FUNCTION_BLOCK SM_DoorDasher EXTENDS KvalStateMachineBaseExt
VAR_INPUT
	cmd_bReset						: BOOL; // reset from error.
	cmd_bCrossTransfer				: BOOL; // true to start cross transfering between 2 adjacent tables.
	cmd_bInlineTransfer				: BOOL; // true to start inline transfering between 2 adjacent tables.
	cmd_bRotateDoor					: BOOL; // true to rotate the door.
	cmd_bCenterDoor					: BOOL; // true to center the door before rotation.
	cmd_bDoorDash					: BOOL; // true to start transport door between adjacent tables.
	cmd_iSource						: INT; // starting table to cross from.
	cmd_iTarget						: INT; // ending table to cross to.
	pstTable						: POINTER TO SM_TableManager;
	pstDoorTrack					: POINTER TO ST_DoorTrack; // pointer to the TableManager's DoorTrack object.
	itfDoorTracker					: I_DoorTracker;
	
	config_tCrossFeedTargetFenceStopEyeValidTime	: TIME := T#20MS;	// time for a valid target fence table's eye.
	
	config_tCrossFeedTargetEyeValidTime	: TIME := T#20MS;	// debouncing time for a valid target table's eye.
	config_tCrossFeedSourceEyeValidTime	: TIME := T#20MS;
	config_tInlineFeedSourceEyeValidTime	: TIME := T#20MS;
	config_tStopMotorValidTime	: TIME := T#30MS;
	
	config_tCrossFeedTargetEyeRisingPreSearchTime	: TIME := T#0.25S;
	config_tInlineFeedTargetEyeRisingPreSearchTime	: TIME := T#0.25S;
	
	config_tCrossFeedTargetEyeRisingPreValidTime	: TIME := T#20MS;
	config_tInlineFeedTargetEyeRisingValidTime	: TIME := T#2.0S;
	
	config_tCrossFeedTargetEyeRisingPostSearchTime	: TIME := T#2.0S;
	config_tInlineFeedTargetEyeRisingPostSearchTime	: TIME := T#2.0S;
	
	config_tCrossFeedTargetEyeRisingPostValidTime	: TIME := T#20MS;
	config_tInlineFeedTargetEyeRisingPostValidTime	: TIME := T#20MS;
	
	config_tCrossFeedTargetEyeRisingPreMaxTime	: TIME := T#3.0S;
	config_tInlineFeedTargetEyeRisingMaxTime	: TIME := T#3.0S;
	
	config_tCrossFeedTargetEyeRisingPostMaxTime	: TIME := T#5.0S;
	config_tInlineFeedTargetEyeFallingMaxTime	: TIME := T#10.0S;
	config_tCrossFeedWaitForAllDoorDashersReady	: TIME := T#0.25S;
	config_tInlineFeedWaitForAllDoorDashersReady	: TIME := T#0.25S;
	config_tCrossFeedSourceEyeRisingSearchTime	: TIME := T#20MS;
	config_tInlineFeedSourceEyeRisingSearchTime	: TIME := T#20MS;
	config_tFindSourceCrossEyeMaxTimeSec		: TIME := T#2.75S; // timeout for finding source's rising edge of feed eye.
	config_tFindSourceInlineEyeMaxTimeSec		: TIME := T#3.5S; // timeout for finding source's rising edge of feed eye.
	config_fFindTargetEyeTimeSec		: LREAL := 12;	// timeout for finding rising or falling edge of the target table's eye. Assumes source and target tables are adjacent neighbors.
	config_fFindRisingEdgeOfTargetFenceEyeTime		: TIME := T#0.25S;
	config_tInlineTargetFeedEyeFallingEdgeTime	: TIME := T#50MS;

	config_iTableArrayIndex			: INT;		// The array table index.
END_VAR
VAR_OUTPUT		
	bMovingFwd					: BOOL; // true if eSource > eTarget
	bIsTargetBufferTable				: BOOL; // used by inline-transfer seq. True to skip the re-feedin seq to center the door on table if the target table is a buffer table with T1 option, which can only inline-transfer and not (cross-transfer or self-center).  
	bIsConveyorAtTarget			: BOOL; // true if the target table is the conveyor type (C235)	
	bIsConveyorAtSource			: BOOL; // true if the source table is the conveyor type (C235)	
	
	bDoorInMachineAtSource		: BOOL;
	bDoorInMachineAtTarget		: BOOL;
	iStopTableIndex : INT;
	bSourceTrailingNeighborDoorDasherBusy : BOOL;
	bSourceLeadingNeighborDoorDasherBusy : BOOL;
	bAllCrossCylsExtended		: BOOL;
	bAllCrossCylsRetracted		: BOOL;
	bOkToTransferOutDoor 		: BOOL;
	bTransferring				: BOOL;
	bCrossTransferSeqRunning	: BOOL;
	bInlineTransferSeqRunning	: BOOL;
	bFoundTarget				: BOOL;
	bAllSourceAndTargetExternal : BOOL;
	bCenteringDoorStarted		: BOOL;
	bCenteringDoorComplete		: BOOL;
	bAnyTableExternal 			: BOOL;
	bSourceTableReady			: BOOL;
	bAllTablesReady				: BOOL;
	bAnyTableBusy				: BOOL;
	sSource						: STRING;
	sTarget						: STRING;
	iSourcePathIndex			: INT;
	iTargetPathIndex			: INT;
	iSourceTrailingNeighborIndex 		: INT;
	iSourceLeadingNeighborIndex 		: INT;
	bStoppingSource : BOOL;
	bStoppingTarget : BOOL;
	bAligningDoorStarted			: BOOL;
	bAligningDoorComplete		: BOOL;
	bFeedingInDoorStarted			: BOOL;
	bFeedingInDoorComplete		: BOOL;
	iNextTarget : INT;
	stNextTargetNode : ST_Node;
	stCurrentTargetNode : ST_Node;
	eNextNodeDirection : E_Direction;
	eSourceTrailingNeighborNodeDirection : E_Direction;
	eSourceLeadingNeighborNodeDirection : E_Direction;
	
	bCrossTransferWaitingForAllDoorDashersReady : BOOL;
	bCrossTransferWaitingForAllDoorDashersComplete : BOOL;
	bInlineTransferWaitingForAllDoorDashersReady : BOOL;
	bInlineTransferWaitingForAllDoorDashersComplete : BOOL;
	
	bCrossTransferSourceTrailingNeighborReady : BOOL;
	bCrossTransferSourceLeadingNeighborReady : BOOL;
	bCrossTransferSourceTrailingNeighborComplete : BOOL;
	bCrossTransferSourceLeadingNeighborComplete : BOOL;
	
	bInlineTransferSourceTrailingNeighborReady : BOOL;
	bInlineTransferSourceLeadingNeighborReady : BOOL;
	bInlineTransferSourceTrailingNeighborComplete : BOOL;
	bInlineTransferSourceLeadingNeighborComplete : BOOL;
END_VAR
VAR CONSTANT
	
END_VAR
VAR
	bTargetTransferTableCandDsideDoorFeedEyesClear : BOOL; // invariant - if the target is a transfer table, its C and D feed eyes must be clear (ie, door is completely in machine) in-order to proceed to next seq. 
	cmd_bReverseDirectionForWideDoor	: BOOL; // true when a wide door (42-in width door) triggers a near/far fence eye as it comes to a stop on falling edge of C/D eye on the C234 feed table.
	pdi_crossSourceFeedEyeRisingEdge					: POINTER TO BOOL; // pointer to the source table's feed eye.
	pdi_crossTargetFeedEyeEdgePre					: POINTER TO BOOL; // cross-transfer pointer to the target table's feed eye.
	pdi_crossTargetFeedEyeRisingEdgePost					: POINTER TO BOOL; // cross-transfer pointer to the target table's feed eye.
	
	pdi_inlineSourceFeedEyeRisingEdge					: POINTER TO BOOL; // inline-transfer pointer to the source table's feed eye.
	pdi_inlineTargetFeedEyeRisingEdge					: POINTER TO BOOL; // inline-transfer pointer to the target table's feed eye rising edge.
	pdi_inlineTargetFeedEyeFallingEdge					: POINTER TO BOOL; // inline-transfer pointer to the target table's feed eye falling edge.

	pdi_targetFenceEye					: POINTER TO BOOL; // pointer to the target table's near/far-fence eye of C234 feed manager.
	pdi_targetFenceStopEye				: POINTER TO BOOL; // pointer to the target table's feed-stop eye, C/D eye of C234 feed manager.
	
	ftrigRotateComplete							: F_TRIG; // trigger to indicate the rotate sequence is completed.
	ftrigSelfCenterComplete						: F_TRIG; // trigger to indicate the self-center sequence is completed.
	ftrigAlignComplete							: F_TRIG; // trigger to indicate the align sequence is completed.
	
	rtrigAllTablesExternal : R_TRIG; // rising edge triggered on all tables are in External state.
	rtrigAllTablesInternal : R_TRIG; // rising edge triggered on all tables are in Internal state.
	rtrigAllTablesCrossCylsExtended : R_TRIG; // rising edge triggered on all tables' cross cylinders are extended.
	rtrigAllTablesCrossCylsRetracted : R_TRIG; // rising edge triggered on all tables' cross cylinders are retracted.
	rtrigAllTablesMotorsMoving : R_TRIG; // rising edge triggered on all tables' VFD motors are moving.
	ftrigAnyTablesMotorsMoving : F_TRIG; // falling edge triggered on all tables' VFD motors are not moving.
	
	rtrigSourceLeadingAndTrailingNeighborsReady : R_TRIG;
	rtrigSourceLeadingAndTrailingNeighborsComplete : R_TRIG;
	rtrigSourceMotorMoving : R_TRIG;
	ftrigSourceMotorMoving : F_TRIG;
	rtrigTargetMotorMoving : R_TRIG;
	ftrigTargetMotorMoving : F_TRIG;
	rtrigSourceFeedEye : R_TRIG;
	rtrigTargetFeedEyePre : R_TRIG;
	rtrigTargetFeedEyePost : R_TRIG;
	
	rtrigInlineSourceFeedEye : R_TRIG;
	rtrigInlineTargetFeedEyeRising : R_TRIG;
	ftrigInlineTargetFeedEyeFalling : F_TRIG;
	
	rtrigTargetCrossFeedEye : R_TRIG; // rising edge triggered on the target table's cross-feed eye.
	ftrigTargetCrossFeedEye : F_TRIG; // falling edge triggered on the target table's cross-feed eye. (for detecting the C234's falling eye)
	
	rtrigCrossTargetFenceStopEye : R_TRIG;
	
	rtrigTargetFenceEye : R_TRIG; // rising edge triggered on the target table's cross- near/far fence eye.
	ftrigAutofeedOn				: F_TRIG; // falling edge of cmd_bAutofeedOn.	
	tonCrossFeedTargetEyeValidTimer				: TON;
	tonCrossFeedSourceEyeValidTimer				: TON;
	tonInlineFeedSourceEyeValidTimer				: TON;
	tonCrossFeedTargetFenceEyeValidTimer				: TON;
	tonCrossFeedTargetStopEyeValidTimer				: TON;
	tofCrossFeedTargetEyeValidTimer			: TOF;
	tofInlineTargetFeedEyeFallingEdgeTimer					: TOF;
	
	tofStopMotorValidTimer			: TOF;
	tonFeedAllDoorDasherReadyTimer				: TON;
	tonFeedTargetEyePreValidTimer				: TON;
	tonFeedTargetEyePostValidTimer				: TON;
tonInlineFeedTargetEyeRisingValidTimer				: TON;
	tFindTargetEyeTimeout						: TIME;
	stTargetPath : ST_PathInfo;
END_VAR

runMachine();

METHOD activateTablesCrossCyls
VAR 
	i : INT;
	tableIndex : INT;
END_VAR
FOR i:=iSourcePathIndex TO iTargetPathIndex DO
	tableIndex := stTargetPath.Path[i].TableIndex;
	IF NOT MAIN.mainStateMachine.asmTableManagers[tableIndex].config_bIsConveyorTable THEN
		MAIN.mainStateMachine.asmTableManagers[tableIndex].smC234FeedManager.cmd_bRaiseCrossCyls := TRUE;
	END_IF
END_FOR
END_METHOD

METHOD alignDoorAtTarget
IF NOT bIsConveyorAtTarget THEN
	MAIN.mainStateMachine.asmTableManagers[cmd_iTarget].smC234FeedManager.cmd_bAlign := TRUE;
END_IF
END_METHOD

METHOD allTablesCrossCylsExtended : BOOL
VAR 
	i : INT;
	tableIndex : INT;
END_VAR
allTablesCrossCylsExtended := TRUE;
FOR i:=iSourcePathIndex TO iTargetPathIndex DO
	tableIndex := stTargetPath.Path[i].TableIndex;
	IF MAIN.mainStateMachine.asmTableManagers[tableIndex].config_bIsBufferTable OR
		MAIN.mainStateMachine.asmTableManagers[tableIndex].config_bIsConveyorTable THEN
		CONTINUE;
	END_IF
	IF NOT MAIN.mainStateMachine.asmTableManagers[tableIndex].smC234FeedManager.bCrossfeedCylsExtended THEN
		allTablesCrossCylsExtended := FALSE;
		RETURN;
	END_IF
END_FOR
END_METHOD

METHOD allTablesCrossCylsRetracted : BOOL
VAR 
	i : INT;
	tableIndex : INT;
END_VAR
allTablesCrossCylsRetracted := TRUE;
FOR i:=iSourcePathIndex TO iTargetPathIndex DO
	tableIndex := stTargetPath.Path[i].TableIndex;
	IF MAIN.mainStateMachine.asmTableManagers[tableIndex].config_bIsBufferTable OR
	 	MAIN.mainStateMachine.asmTableManagers[tableIndex].config_bIsConveyorTable THEN
		CONTINUE;
	END_IF
	IF NOT MAIN.mainStateMachine.asmTableManagers[tableIndex].smC234FeedManager.bCrossfeedCylsRetracted THEN
		allTablesCrossCylsRetracted := FALSE;
		RETURN;
	END_IF
END_FOR
END_METHOD

METHOD allTablesExternal : BOOL
VAR 
	i : INT;
	tableIndex : INT;
END_VAR
allTablesExternal := TRUE;
FOR i:=iSourcePathIndex TO iTargetPathIndex DO
	tableIndex := stTargetPath.Path[i].TableIndex;
	IF NOT MAIN.mainStateMachine.asmTableManagers[tableIndex].bExternal THEN
		allTablesExternal := FALSE;
		RETURN;
	END_IF
END_FOR
END_METHOD

METHOD allTablesMotorsMoving : BOOL
VAR 
	i : INT;
	tableIndex : INT;
END_VAR
allTablesMotorsMoving := TRUE;
FOR i:=iSourcePathIndex TO iTargetPathIndex DO
	tableIndex := stTargetPath.Path[i].TableIndex;
	IF NOT MAIN.mainStateMachine.asmTableManagers[tableIndex].status_bMoving THEN
		allTablesMotorsMoving := FALSE;
		RETURN;
	END_IF
END_FOR
END_METHOD

METHOD anyTableBusy : BOOL
VAR 
	i : INT;
	tableIndex : INT;
END_VAR
anyTableBusy := FALSE;
FOR i:=iSourcePathIndex TO iTargetPathIndex DO
	tableIndex := stTargetPath.Path[i].TableIndex;
	IF MAIN.mainStateMachine.asmTableManagers[tableIndex].anyChildBusy() THEN
		anyTableBusy := TRUE;
		RETURN;
	END_IF
END_FOR
END_METHOD

METHOD anyTableExternal : BOOL
VAR 
	i : INT;
	tableIndex : INT;
END_VAR
anyTableExternal := FALSE;
FOR i:=iSourcePathIndex TO iTargetPathIndex DO
	tableIndex := stTargetPath.Path[i].TableIndex;
	IF MAIN.mainStateMachine.asmTableManagers[tableIndex].bExternal THEN
		anyTableExternal := TRUE;
		RETURN;
	END_IF
END_FOR
END_METHOD

METHOD anyTableMotorMoving : BOOL
VAR 
	i : INT;
	tableIndex : INT;
END_VAR
anyTableMotorMoving := FALSE;

IF cmd_iSource <> cmd_iTarget THEN
	FOR i:=iSourcePathIndex TO iTargetPathIndex DO
		tableIndex := stTargetPath.Path[i].TableIndex;
		IF tableIndex = cmd_iSource THEN
			IF bStoppingSource AND MAIN.mainStateMachine.asmTableManagers[tableIndex].status_bMoving THEN
				anyTableMotorMoving := TRUE;
				RETURN;
			END_IF
		ELSE
			IF bStoppingTarget AND MAIN.mainStateMachine.asmTableManagers[tableIndex].status_bMoving THEN
				anyTableMotorMoving := TRUE;
				RETURN;
			END_IF
		END_IF
	END_FOR
END_IF
END_METHOD

METHOD areTablesReady : BOOL
VAR 
	i : INT;
	tableIndex : INT;
END_VAR
areTablesReady := TRUE;
FOR i:=iSourcePathIndex TO iTargetPathIndex DO
	tableIndex := stTargetPath.Path[i].TableIndex;
	IF MAIN.mainStateMachine.asmTableManagers[tableIndex].anyChildBusy() OR 
		NOT MAIN.mainStateMachine.asmTableManagers[tableIndex].cmd_bAutoFeedOn OR 
		MAIN.mainStateMachine.asmTableManagers[tableIndex].bExternal THEN
		areTablesReady := FALSE;
		RETURN;
	END_IF
END_FOR
END_METHOD

METHOD centerDoorAtSource
IF NOT bIsConveyorAtSource AND MAIN.mainStateMachine.asmTableManagers[cmd_iSource].config_bCanSelfCenter THEN
	MAIN.mainStateMachine.asmTableManagers[cmd_iSource].smC234FeedManager.smSelfCenterManager.cmd_bSelfCenter := TRUE;
END_IF
END_METHOD

METHOD crossFast
VAR 
	i : INT;
	tableIndex : INT;
END_VAR
FOR i:=iSourcePathIndex TO iTargetPathIndex DO
	tableIndex := stTargetPath.Path[i].TableIndex;
	MAIN.mainStateMachine.asmTableManagers[tableIndex].psmHcFeedMotor^.cmd_iSpeedRPM := MAIN.mainStateMachine.asmTableManagers[tableIndex].iCrossFeedFastSpeedRPM;
END_FOR
END_METHOD

METHOD crossFwd
VAR 
	i : INT;
	tableIndex : INT;
END_VAR
FOR i:=iSourcePathIndex TO iTargetPathIndex DO
	tableIndex := stTargetPath.Path[i].TableIndex;
	IF MAIN.mainStateMachine.asmTableManagers[tableIndex].config_bIsConveyorTable THEN
		MAIN.mainStateMachine.asmTableManagers[tableIndex].goFwd();
	ELSE
		// inverted direction when crossing for the C234 feed.
		MAIN.mainStateMachine.asmTableManagers[tableIndex].goRev();
	END_IF
		
END_FOR
END_METHOD

METHOD crossRev
VAR 
	i : INT;
	tableIndex : INT;
END_VAR
FOR i:=iSourcePathIndex TO iTargetPathIndex DO
	tableIndex := stTargetPath.Path[i].TableIndex;
	IF MAIN.mainStateMachine.asmTableManagers[tableIndex].config_bIsConveyorTable THEN
		MAIN.mainStateMachine.asmTableManagers[tableIndex].goRev();
	ELSE
		// inverted direction when crossing for the C234 feed.
		MAIN.mainStateMachine.asmTableManagers[tableIndex].goFwd();
	END_IF
		
END_FOR
END_METHOD

METHOD crossSlow
VAR 
	i : INT;
	tableIndex : INT;
END_VAR
FOR i:=iSourcePathIndex TO iTargetPathIndex DO
	tableIndex := stTargetPath.Path[i].TableIndex;
	MAIN.mainStateMachine.asmTableManagers[tableIndex].psmHcFeedMotor^.cmd_iSpeedRPM := MAIN.mainStateMachine.asmTableManagers[tableIndex].iCrossFeedSlowSpeedRPM;
END_FOR
END_METHOD

METHOD crossSlower
VAR 
	i : INT;
	tableIndex : INT;
END_VAR
FOR i:=iSourcePathIndex TO iTargetPathIndex DO
	tableIndex := stTargetPath.Path[i].TableIndex;
	MAIN.mainStateMachine.asmTableManagers[tableIndex].psmHcFeedMotor^.cmd_iSpeedRPM := MAIN.mainStateMachine.asmTableManagers[tableIndex].iCrossFeedSlowSpeedRPM/2;
END_FOR
END_METHOD

METHOD crossTransferStart
tFindTargetEyeTimeout := LREAL_TO_TIME((ABS(iSourcePathIndex - iTargetPathIndex) * config_fFindTargetEyeTimeSec) * 1000);
sSource := getTableName(cmd_iSource);
sTarget := getTableName(cmd_iTarget);
bIsConveyorAtTarget := MAIN.mainStateMachine.asmTableManagers[cmd_iTarget].config_bIsConveyorTable;
bIsConveyorAtSource := MAIN.mainStateMachine.asmTableManagers[cmd_iSource].config_bIsConveyorTable;
bDoorInMachineAtSource		:= MAIN.mainStateMachine.asmTableManagers[cmd_iSource].bDoorInMachine;
bDoorInMachineAtTarget		:= MAIN.mainStateMachine.asmTableManagers[cmd_iTarget].bDoorInMachine;
MAIN.mainStateMachine.asmTableManagers[cmd_iSource].setTransferOutStarted();
MAIN.mainStateMachine.asmTableManagers[cmd_iTarget].setDoorTransferredInStarted();

IF bIsConveyorAtSource THEN
	IF bMovingFwd THEN
		pdi_crossSourceFeedEyeRisingEdge := ADR( MAIN.mainStateMachine.asmTableManagers[cmd_iSource].smC235FeedManager.di_CSideDoorFeedEye);
	ELSE
		pdi_crossSourceFeedEyeRisingEdge := ADR( MAIN.mainStateMachine.asmTableManagers[cmd_iSource].smC235FeedManager.di_DSideDoorFeedEye);
	END_IF
ELSE
	IF bMovingFwd THEN
		pdi_crossSourceFeedEyeRisingEdge := ADR( MAIN.mainStateMachine.asmTableManagers[cmd_iSource].smC234FeedManager.di_CSideDoorFeedEye);
	ELSE
		pdi_crossSourceFeedEyeRisingEdge := ADR( MAIN.mainStateMachine.asmTableManagers[cmd_iSource].smC234FeedManager.di_DSideDoorFeedEye);
	END_IF
END_IF

IF bIsConveyorAtTarget THEN
	IF bMovingFwd THEN
		pdi_crossTargetFeedEyeEdgePre := ADR( MAIN.mainStateMachine.asmTableManagers[cmd_iTarget].smC235FeedManager.di_DSideDoorFeedEye);
		pdi_crossTargetFeedEyeRisingEdgePost := ADR( MAIN.mainStateMachine.asmTableManagers[cmd_iTarget].smC235FeedManager.di_CSideDoorFeedEye);
	ELSE
		pdi_crossTargetFeedEyeEdgePre := ADR( MAIN.mainStateMachine.asmTableManagers[cmd_iTarget].smC235FeedManager.di_CSideDoorFeedEye);
		pdi_crossTargetFeedEyeRisingEdgePost := ADR( MAIN.mainStateMachine.asmTableManagers[cmd_iTarget].smC235FeedManager.di_DSideDoorFeedEye);
	END_IF
ELSE
	IF bMovingFwd THEN
		pdi_crossTargetFeedEyeEdgePre := ADR( MAIN.mainStateMachine.asmTableManagers[cmd_iTarget].smC234FeedManager.di_DSideDoorFeedEye);
		pdi_targetFenceEye := ADR(MAIN.mainStateMachine.asmTableManagers[cmd_iTarget].smC234FeedManager.di_AtFarFenceEye);
		pdi_targetFenceStopEye := ADR(MAIN.mainStateMachine.asmTableManagers[cmd_iTarget].smC234FeedManager.di_AtNearFenceEye);
	ELSE
		pdi_crossTargetFeedEyeEdgePre := ADR( MAIN.mainStateMachine.asmTableManagers[cmd_iTarget].smC234FeedManager.di_CSideDoorFeedEye);
		pdi_targetFenceEye := ADR(MAIN.mainStateMachine.asmTableManagers[cmd_iTarget].smC234FeedManager.di_AtNearFenceEye);
		pdi_targetFenceStopEye := ADR(MAIN.mainStateMachine.asmTableManagers[cmd_iTarget].smC234FeedManager.di_AtFarFenceEye);
	END_IF
END_IF
END_METHOD

METHOD deactivateTablesCrossCyls
VAR 
	i : INT;
	tableIndex : INT;
END_VAR
FOR i:=iSourcePathIndex TO iTargetPathIndex DO
	tableIndex := stTargetPath.Path[i].TableIndex;
	IF NOT MAIN.mainStateMachine.asmTableManagers[tableIndex].config_bIsConveyorTable THEN
		MAIN.mainStateMachine.asmTableManagers[tableIndex].smC234FeedManager.cmd_bLowerCrossCyls := TRUE;
	END_IF
END_FOR
END_METHOD

METHOD doorDash
VAR
	i : INT;
	j : INT;	
END_VAR
stCurrentTargetNode := stNodeDefault;
stNextTargetNode := stNodeDefault;
cmd_bRotateDoor := FALSE;
cmd_bCenterDoor := FALSE;
cmd_bCrossTransfer := FALSE;
cmd_bInlineTransfer := FALSE;
bOkToTransferOutDoor := FALSE;
stTargetPath := stPathInfoDefault;
eSourceTrailingNeighborNodeDirection := E_Direction.None;
eSourceLeadingNeighborNodeDirection := E_Direction.None;

FOR i:= 0 TO pstDoorTrack^.TargetPath.PathCount - 1 DO
	// do we have the source from TargetPath?
	IF pstDoorTrack^.TargetPath.Path[i].TableIndex = config_iTableArrayIndex THEN
		// found the source in TargetPath
		stCurrentTargetNode := pstDoorTrack^.TargetPath.Path[i];
		cmd_iSource := stCurrentTargetNode.TableIndex;
		cmd_iTarget := cmd_iSource; // set the target as the same as source.
		stTargetPath := pstDoorTrack^.TargetPath;
		
		IF stCurrentTargetNode.Direction <> E_Direction.None THEN
			// do we have the target in TargetPath? 
			iNextTarget := i + 1;
			IF iNextTarget < pstDoorTrack^.TargetPath.PathCount THEN
				// found the target in TargetPath
				FOR j:= iNextTarget TO pstDoorTrack^.TargetPath.PathCount - 1 DO
					stNextTargetNode := pstDoorTrack^.TargetPath.Path[j];
					eNextNodeDirection := MAIN.mainStateMachine.asmTableManagers[stNextTargetNode.TableIndex].getTargetNodeDirection();
					IF MAIN.mainStateMachine.asmTableManagers[stNextTargetNode.TableIndex].bExternal OR 
						MAIN.mainStateMachine.asmTableManagers[stNextTargetNode.TableIndex].bFindingPath OR
						MAIN.mainStateMachine.asmTableManagers[stNextTargetNode.TableIndex].bRouteReadyWaitForFeedIn OR
						MAIN.mainStateMachine.asmTableManagers[stNextTargetNode.TableIndex].bWaitAllTablesReady OR
						MAIN.mainStateMachine.asmTableManagers[stNextTargetNode.TableIndex].bDoorWaitingForFeedOut OR
						MAIN.mainStateMachine.asmTableManagers[stNextTargetNode.TableIndex].bDoorFeedingOut OR
						MAIN.mainStateMachine.asmTableManagers[stNextTargetNode.TableIndex].status_bBusy OR
						(eNextNodeDirection <> E_Direction.None AND stCurrentTargetNode.Direction <> eNextNodeDirection) THEN
						// do not run DoorDasher seq if the target is external and being controlled by the target's DoorDasher seq.
						EXIT;
					ELSIF  
						NOT 
							// any of these is true, the target has a door already in machine or new incoming door, we keep searching until we found a table without door.   
							(MAIN.mainStateMachine.asmTableManagers[stNextTargetNode.TableIndex].bHasDoor OR 
							(MAIN.mainStateMachine.asmTableManagers[stNextTargetNode.TableIndex].cmd_bDoorDataReadyLatched XOR
							MAIN.mainStateMachine.asmTableManagers[stNextTargetNode.TableIndex].bWaitingForClearRoute) OR 
							MAIN.mainStateMachine.asmTableManagers[stNextTargetNode.TableIndex].bRouteReadyWaitForFeedIn OR							
							MAIN.mainStateMachine.asmTableManagers[stNextTargetNode.TableIndex].bDoorFeedingIn OR
							MAIN.mainStateMachine.asmTableManagers[stNextTargetNode.TableIndex].bDoorInMachineIdle OR
							MAIN.mainStateMachine.asmTableManagers[stNextTargetNode.TableIndex].bDoorWaitingForFeedOut
							) THEN
						bOkToTransferOutDoor := MAIN.mainStateMachine.asmTableManagers[stNextTargetNode.TableIndex].bWaitForDataReadyOrTransferredIn;
						EXIT;
					ELSE
						IF stCurrentTargetNode.Direction = eNextNodeDirection THEN
							CONTINUE;
						END_IF
					END_IF
				END_FOR
			END_IF
		END_IF		
		EXIT;
	END_IF
END_FOR

IF bOkToTransferOutDoor THEN
	bMovingFwd := 
		stCurrentTargetNode.Direction = E_Direction.North
		OR stCurrentTargetNode.Direction = E_Direction.East 
		;
	stNextTargetNode := pstDoorTrack^.TargetPath.Path[iNextTarget];
	cmd_iTarget := stNextTargetNode.TableIndex;
	
	cmd_bCrossTransfer := stCurrentTargetNode.Direction = E_Direction.North OR stCurrentTargetNode.Direction = E_Direction.South;
	cmd_bInlineTransfer := stCurrentTargetNode.Direction = E_Direction.West OR stCurrentTargetNode.Direction = E_Direction.East;	
END_IF

cmd_bRotateDoor := 
	 pstTable^.smC234FeedManager.config_bCanRotate AND 
	 pstTable^.smC234FeedManager.config_bCanSelfCenter AND
	(pstDoorTrack^.DoorRotateRequired XOR pstDoorTrack^.DoorWasRotated)	
; 	

cmd_bCenterDoor := cmd_bRotateDoor AND pstTable^.smC234FeedManager.config_eFeedoutAligned <> E_FeedoutAligned.CenterFence;
cmd_bDoorDash := 
	cmd_bCrossTransfer OR
	cmd_bInlineTransfer OR
	cmd_bRotateDoor;

bTransferring := 
	cmd_bCrossTransfer OR
	cmd_bInlineTransfer;
	
IF bTransferring THEN
	iSourceTrailingNeighborIndex := findSourceTrailingNeighborTableIndex();
	iSourceLeadingNeighborIndex := findSourceLeadingNeighborTableIndex();

	IF iSourceTrailingNeighborIndex <> -1 THEN
		eSourceTrailingNeighborNodeDirection :=  MAIN.mainStateMachine.asmTableManagers[iSourceTrailingNeighborIndex].getTargetNodeDirection();
	END_IF
	IF iSourceLeadingNeighborIndex <> -1 THEN
		eSourceLeadingNeighborNodeDirection :=  MAIN.mainStateMachine.asmTableManagers[iSourceLeadingNeighborIndex].getTargetNodeDirection();
	END_IF
END_IF
	
IF cmd_bDoorDash THEN
	status_bBusy := TRUE; // set busy here to prevent triggerring door-dasher seq again.
	iSourcePathIndex := findTargetPathIndex(cmd_iSource);
	iTargetPathIndex := findTargetPathIndex(cmd_iTarget);
END_IF
END_METHOD

METHOD doState
CASE (machineState) OF	
	DOOR_DASHER_DISABLED:
		IF bFirstPass THEN
		   downstream.setAllDownstreamDisabled();
			status_bReady := FALSE;
			status_bBusy := FALSE;
			bCrossTransferSeqRunning	:= FALSE;
			bInlineTransferSeqRunning	:= FALSE;
			bTransferring := FALSE;
		END_IF

	DOOR_DASHER_ENABLING:
		IF bFirstPass THEN
			 downstream.setAllDownstreamEnabled();
		END_IF
		IF downstream.status_bDownstreamAllReady THEN
			machineState := DOOR_DASHER_AUTOFEED_OFF;
		END_IF
	
	DOOR_DASHER_AUTOFEED_OFF:
		IF bFirstPass THEN
			status_bReady := TRUE;
			status_bBusy := FALSE;
			bAllTablesReady := FALSE;
			bAllSourceAndTargetExternal := FALSE;
			bCrossTransferSeqRunning	:= FALSE;
			bInlineTransferSeqRunning	:= FALSE;
			bTransferring := FALSE;
			stop();
		END_IF
		IF cmd_bAutoFeedOn THEN
			machineState := DOOR_DASHER_AUTOFEED_ON;
		END_IF
		
	DOOR_DASHER_AUTOFEED_ON:
        IF bFirstPass THEN
			status_bBusy := FALSE;
			bAllTablesReady := FALSE;
			bAllSourceAndTargetExternal := FALSE;
			bCrossTransferSeqRunning	:= FALSE;
			bInlineTransferSeqRunning	:= FALSE;
			bTransferring := FALSE;
			stop();
		END_IF
		IF NOT cmd_bAutoFeedOn THEN
			machineState := DOOR_DASHER_AUTOFEED_OFF;
        ELSIF cmd_bDoorDash THEN
			machineState := DOOR_DASHER_START;
		END_IF

	DOOR_DASHER_START:
		IF bFirstPass THEN
			bFoundTarget := FALSE;
			bAllTablesReady := FALSE;
			bSourceTableReady := FALSE;
			bAllSourceAndTargetExternal := FALSE;
		ELSIF cmd_bNext THEN
			machineState := DOOR_DASHER_WAIT_FOR_SOURCE_TABLE_READY;
		END_IF
		
	DOOR_DASHER_WAIT_FOR_SOURCE_TABLE_READY:
		IF bFirstPass THEN
			;
		END_IF
		bSourceTableReady := isSourceTableReady();
		IF bSourceTableReady THEN
			machineState := DOOR_DASHER_WAIT_FOR_SOURCE_AND_TARGET_EXTERNAL;
		END_IF
	
	DOOR_DASHER_WAIT_FOR_SOURCE_AND_TARGET_EXTERNAL:
        IF bFirstPass THEN
			setExternal();
		ELSE
			bAllSourceAndTargetExternal := allTablesExternal();
			IF bAllSourceAndTargetExternal THEN
				IF cmd_bCenterDoor THEN
					machineState := DOOR_DASHER_CENTER_DOOR_PRE_ROTATE;
				ELSIF cmd_bRotateDoor THEN
					machineState := DOOR_DASHER_ROTATE_DOOR;
				ELSE
					machineState := DOOR_DASHER_READY_TO_TRANSFER;
				END_IF
			END_IF
		END_IF
	
	DOOR_DASHER_CENTER_DOOR_PRE_ROTATE:
		IF bFirstPass THEN
			pstTable^.smC234FeedManager.cmd_bSelfCenter := TRUE;			
		END_IF
		ftrigSelfCenterComplete(CLK:=pstTable^.smC234FeedManager.status_bBusy);
		IF ftrigSelfCenterComplete.Q THEN
			machineState := DOOR_DASHER_ROTATE_DOOR;
		END_IF
		
	DOOR_DASHER_ROTATE_DOOR:
		IF bFirstPass THEN
			pstTable^.smC234FeedManager.cmd_bRotate := TRUE;
			pstDoorTrack^.DoorIsRotating := TRUE;
		END_IF
		ftrigRotateComplete(CLK:=pstTable^.smC234FeedManager.status_bBusy);
		IF ftrigRotateComplete.Q THEN			
			machineState := DOOR_DASHER_ALIGN_DOOR;
		END_IF
	
	DOOR_DASHER_ALIGN_DOOR:
		IF bFirstPass THEN
			pstTable^.smC234FeedManager.cmd_bAlign := TRUE;
		END_IF
		ftrigAlignComplete(CLK:=pstTable^.smC234FeedManager.status_bBusy);
		IF ftrigAlignComplete.Q THEN
			pstDoorTrack^.DoorWasRotated := NOT pstDoorTrack^.DoorWasRotated;
			pstDoorTrack^.DoorIsRotating := FALSE;
			machineState := DOOR_DASHER_READY_TO_TRANSFER;
		END_IF
	
	DOOR_DASHER_READY_TO_TRANSFER:
		IF bFirstPass THEN
			;
		ELSIF cmd_bNext THEN
			IF cmd_bCrossTransfer THEN
				machineState := DOOR_DASHER_CROSS_TRANSFER_START;
			ELSIF cmd_bInlineTransfer THEN
				machineState := DOOR_DASHER_INLINE_TRANSFER_START;
			ELSE
				machineState := DOOR_DASHER_SET_SOURCE_AND_TARGET_INTERNAL;
			END_IF
		END_IF
	
	DOOR_DASHER_CROSS_TRANSFER_START:
        IF bFirstPass THEN			
			crossTransferStart();
			bCrossTransferSeqRunning	:= TRUE;
			cmd_bReverseDirectionForWideDoor := FALSE;
			bAllSourceAndTargetExternal := FALSE;
			bAligningDoorStarted := FALSE;
			bAligningDoorComplete := FALSE;
			bAllCrossCylsExtended := FALSE;
			rtrigTargetCrossFeedEye(CLK:=FALSE);
			ftrigTargetCrossFeedEye(CLK:=FALSE);
			rtrigTargetFenceEye(CLK:=FALSE);
			rtrigSourceFeedEye(CLK:=FALSE);
			rtrigTargetFeedEyePre(CLK:=FALSE);
			rtrigTargetFeedEyePost(CLK:=FALSE);
			tonCrossFeedTargetEyeValidTimer(IN:=FALSE, PT:=config_tCrossFeedTargetEyeValidTime);
			tonCrossFeedSourceEyeValidTimer(IN:=FALSE, PT:=config_tCrossFeedSourceEyeValidTime);
			tonCrossFeedTargetFenceEyeValidTimer(IN:=FALSE, PT:=config_tCrossFeedTargetEyeValidTime);
			tonCrossFeedTargetStopEyeValidTimer(IN:=FALSE, PT:=config_tCrossFeedTargetEyeValidTime);
			tofCrossFeedTargetEyeValidTimer(IN:=FALSE, PT:=config_tCrossFeedTargetEyeValidTime);
		ELSE
			IF bIsConveyorAtSource AND bIsConveyorAtTarget THEN
				// both source and target tables are conveyors.
				IF pdi_crossSourceFeedEyeRisingEdge^ THEN
					// door is on the source' staging/starting eye, go straight to wait for all other trailing and leading neighboring tables to be ready.
					machineState := DOOR_DASHER_CROSS_TRANSFER_WAIT_FOR_ALL_DOORDASHERS_READY;
				ELSE
					// door is not on the source' staging/starting eye, start motor and look for it.
					machineState := DOOR_DASHER_CROSS_TRANSFER_START_SOURCE_MOTOR;	
				END_IF
			ELSIF cmd_bNext THEN
				// either or both source and target tables are inline-transfer tables. So activate their cross cyls.
				machineState := DOOR_DASHER_CROSS_TRANSFER_ACTIVATE_CROSS_CYLS;	
			END_IF
		END_IF

	DOOR_DASHER_CROSS_TRANSFER_ACTIVATE_CROSS_CYLS:
        IF bFirstPass THEN
			activateTablesCrossCyls();
		END_IF
		bAllCrossCylsExtended := allTablesCrossCylsExtended();
        IF bAllCrossCylsExtended OR (config_bNoHardwareTestMode AND tTimeInState>T#0.25S) THEN
			IF pdi_crossSourceFeedEyeRisingEdge^ THEN
				machineState := DOOR_DASHER_CROSS_TRANSFER_WAIT_FOR_ALL_DOORDASHERS_READY;
			ELSE
				machineState := DOOR_DASHER_CROSS_TRANSFER_START_SOURCE_MOTOR;
			END_IF
		END_IF

	DOOR_DASHER_CROSS_TRANSFER_START_SOURCE_MOTOR:
		IF bFirstPass THEN
			IF bMovingFwd THEN
				sourceCrossFwd();
			ELSE
				sourceCrossRev();
			END_IF
			sourceCrossFast();
			rtrigSourceMotorMoving(CLK:=FALSE);
		ELSE
			rtrigSourceMotorMoving(CLK:=isSourceMotorMoving());
			IF rtrigSourceMotorMoving.Q OR (config_bNoHardwareTestMode AND tTimeInState>T#0.25S) THEN
				machineState := DOOR_DASHER_CROSS_TRANSFER_FIND_SOURCE_EYE_RISING_EDGE;
			END_IF
		END_IF
		
	DOOR_DASHER_CROSS_TRANSFER_FIND_SOURCE_EYE_RISING_EDGE:
		IF bFirstPass THEN
			rtrigSourceFeedEye(CLK:=FALSE);
			tonCrossFeedSourceEyeValidTimer(IN:=FALSE, PT:=config_tCrossFeedSourceEyeValidTime);
		ELSE
			tonCrossFeedSourceEyeValidTimer(IN:=pdi_crossSourceFeedEyeRisingEdge^);
			rtrigSourceFeedEye(CLK:=
				tTimeInState > config_tCrossFeedSourceEyeRisingSearchTime AND
				tonCrossFeedSourceEyeValidTimer.Q);
			IF rtrigSourceFeedEye.Q OR (config_bNoHardwareTestMode AND tTimeInState>T#0.25S) THEN
				machineState := DOOR_DASHER_CROSS_TRANSFER_STOP_SOURCE_MOTOR;
			ELSIF tTimeInState > config_tFindSourceCrossEyeMaxTimeSec THEN
				IF bMovingFwd THEN
					iErrorId := DOOR_DASHER_FAILED_TO_FIND_SOURCE_C_EYE_RISING_EDGE;
				ELSE
					iErrorId := DOOR_DASHER_FAILED_TO_FIND_SOURCE_D_EYE_RISING_EDGE;
				END_IF
			END_IF
		END_IF
	
	DOOR_DASHER_CROSS_TRANSFER_STOP_SOURCE_MOTOR:
		IF bFirstPass THEN
			sourceStop();
			ftrigSourceMotorMoving(CLK:=FALSE);
		ELSE
			ftrigSourceMotorMoving(CLK:=isSourceMotorMoving());
			IF ftrigSourceMotorMoving.Q OR (config_bNoHardwareTestMode AND tTimeInState>T#0.25S) THEN
				machineState := DOOR_DASHER_CROSS_TRANSFER_WAIT_FOR_ALL_DOORDASHERS_READY;
			END_IF
		END_IF
	
	DOOR_DASHER_CROSS_TRANSFER_WAIT_FOR_ALL_DOORDASHERS_READY:
		IF bFirstPass THEN
			rtrigSourceLeadingAndTrailingNeighborsReady(CLK:=FALSE);
			bCrossTransferSourceTrailingNeighborReady := FALSE;
			bCrossTransferSourceLeadingNeighborReady := FALSE;
		ELSE
			IF NOT bCrossTransferSourceTrailingNeighborReady THEN
				bCrossTransferSourceTrailingNeighborReady := isSourceTrailingNeighborReady();
			END_IF
			IF NOT bCrossTransferSourceLeadingNeighborReady THEN
				bCrossTransferSourceLeadingNeighborReady := isSourceLeadingNeighborReady();
			END_IF
			rtrigSourceLeadingAndTrailingNeighborsReady(CLK:=
				cmd_bNext AND
				bCrossTransferSourceLeadingNeighborReady AND 
				bCrossTransferSourceTrailingNeighborReady
				);
			IF rtrigSourceLeadingAndTrailingNeighborsReady.Q THEN
				machineState := DOOR_DASHER_CROSS_TRANSFER_START_MOTORS;
			END_IF
		END_IF
				
	DOOR_DASHER_CROSS_TRANSFER_START_MOTORS:
        IF bFirstPass THEN
			IF bMovingFwd THEN
				crossFwd();
			ELSE
				crossRev();
			END_IF
			crossFast();
			rtrigAllTablesMotorsMoving(CLK:=FALSE);
			rtrigSourceFeedEye(CLK:=FALSE);
		ELSE
			rtrigAllTablesMotorsMoving(CLK:=allTablesMotorsMoving());
			IF rtrigAllTablesMotorsMoving.Q OR (config_bNoHardwareTestMode AND tTimeInState>T#5.25S) THEN
				machineState := DOOR_DASHER_CROSS_TRANSFER_FIND_TARGET_EYE_RISING_EDGE_PRE;
			END_IF
		END_IF

	DOOR_DASHER_CROSS_TRANSFER_FIND_TARGET_EYE_RISING_EDGE_PRE:
		IF bFirstPass THEN
			rtrigTargetFeedEyePre(CLK:=FALSE);
			tonFeedTargetEyePreValidTimer(IN:=FALSE, PT:=config_tCrossFeedTargetEyeRisingPreValidTime);
		ELSE
			tonFeedTargetEyePreValidTimer(IN:=pdi_crossTargetFeedEyeEdgePre^);
			rtrigTargetFeedEyePre(CLK:=
				tTimeInState > config_tCrossFeedTargetEyeRisingPreSearchTime AND 
				tonFeedTargetEyePreValidTimer.Q);
			IF rtrigTargetFeedEyePre.Q OR (config_bNoHardwareTestMode AND tTimeInState>T#0.25S) THEN
				IF bIsConveyorAtTarget THEN
					machineState := DOOR_DASHER_CROSS_TRANSFER_FIND_TARGET_EYE_RISING_EDGE_POST;
				ELSE
					machineState := DOOR_DASHER_CROSS_TRANSFER_FIND_RISING_OR_FALLING_EDGE_OF_TARGET_EYE;
				END_IF
			ELSIF tTimeInState > config_tCrossFeedTargetEyeRisingPreMaxTime THEN
				IF bMovingFwd THEN
					iErrorId := DOOR_DASHER_FAILED_TO_FIND_TARGET_D_EYE_RISING_EDGE;
				ELSE
					iErrorId := DOOR_DASHER_FAILED_TO_FIND_TARGET_C_EYE_RISING_EDGE;
				END_IF
			END_IF
		END_IF
		
	DOOR_DASHER_CROSS_TRANSFER_FIND_TARGET_EYE_RISING_EDGE_POST:
		IF bFirstPass THEN
			rtrigTargetFeedEyePost(CLK:=FALSE);
			tonFeedTargetEyePostValidTimer(IN:=FALSE, PT:=config_tCrossFeedTargetEyeRisingPostValidTime);
		ELSE
			tonFeedTargetEyePostValidTimer(IN:=pdi_crossTargetFeedEyeRisingEdgePost^);
			rtrigTargetFeedEyePost(CLK:=
				tTimeInState > config_tCrossFeedTargetEyeRisingPostSearchTime AND 
				tonFeedTargetEyePostValidTimer.Q);
			IF rtrigTargetFeedEyePost.Q OR (config_bNoHardwareTestMode AND tTimeInState>T#0.25S) THEN
				machineState := DOOR_DASHER_CROSS_TRANSFER_STOP_MOTORS;
			ELSIF tTimeInState > config_tCrossFeedTargetEyeRisingPostMaxTime THEN
				IF bMovingFwd THEN
					iErrorId := DOOR_DASHER_FAILED_TO_FIND_TARGET_C_EYE_RISING_EDGE;
				ELSE
					iErrorId := DOOR_DASHER_FAILED_TO_FIND_TARGET_D_EYE_RISING_EDGE;
				END_IF
			END_IF
		END_IF
	
	DOOR_DASHER_CROSS_TRANSFER_FIND_RISING_OR_FALLING_EDGE_OF_TARGET_EYE:
        IF bFirstPass THEN
			rtrigTargetCrossFeedEye(CLK:=FALSE);
			ftrigTargetCrossFeedEye(CLK:=FALSE);
			rtrigTargetFenceEye(CLK:=FALSE);
			tonCrossFeedTargetEyeValidTimer(IN:=FALSE, PT:=config_tCrossFeedTargetEyeValidTime);
			tonCrossFeedTargetFenceEyeValidTimer(IN:=FALSE, PT:=config_tCrossFeedTargetEyeValidTime);
			tonCrossFeedTargetStopEyeValidTimer(IN:=FALSE, PT:=config_tCrossFeedTargetEyeValidTime);
			tofCrossFeedTargetEyeValidTimer(IN:=FALSE, PT:=config_tCrossFeedTargetEyeValidTime);
		ELSE
			tonCrossFeedTargetFenceEyeValidTimer(IN:=pdi_targetFenceEye^);
			tofCrossFeedTargetEyeValidTimer(IN:=pdi_crossTargetFeedEyeEdgePre^);
			rtrigTargetFenceEye(CLK:=tonCrossFeedTargetFenceEyeValidTimer.Q);
			ftrigTargetCrossFeedEye(CLK:=tofCrossFeedTargetEyeValidTimer.Q);
			IF rtrigTargetCrossFeedEye.Q OR 
				ftrigTargetCrossFeedEye.Q OR
				(config_bNoHardwareTestMode AND tTimeInState>T#0.25S) THEN
				machineState := DOOR_DASHER_CROSS_TRANSFER_STOP_MOTORS;
			ELSIF tTimeInState > tFindTargetEyeTimeout THEN
				iErrorId := DOOR_DASHER_FAILED_TO_FIND_FALLING_EDGE_OF_TARGET_FEED_EYE_OR_RISING_EDGE_FENCE_EYE;
			END_IF
		END_IF
	
	DOOR_DASHER_CROSS_TRANSFER_STOP_MOTORS:
        IF bFirstPass THEN
			stop();
			ftrigAnyTablesMotorsMoving(CLK:=FALSE);
			tonCrossFeedTargetFenceEyeValidTimer(IN:=FALSE, PT:=config_tCrossFeedTargetEyeValidTime);
			tofStopMotorValidTimer(IN:=FALSE, PT:=config_tStopMotorValidTime);
			rtrigTargetFenceEye(CLK:=FALSE);
			cmd_bReverseDirectionForWideDoor := FALSE;
		ELSE
			tofStopMotorValidTimer(IN:=anyTableMotorMoving());
			ftrigAnyTablesMotorsMoving(CLK:=tofStopMotorValidTimer.Q);
			IF NOT bIsConveyorAtTarget AND pdi_targetFenceEye <> 0 THEN
				tonCrossFeedTargetFenceEyeValidTimer(IN:=pdi_targetFenceEye^, PT:=config_tCrossFeedTargetEyeValidTime);
				rtrigTargetFenceEye(CLK:=tonCrossFeedTargetFenceEyeValidTimer.Q);
				IF rtrigTargetFenceEye.Q OR (config_bNoHardwareTestMode AND tTimeInState>T#0.25S) THEN
					cmd_bReverseDirectionForWideDoor := TRUE;
				END_IF
			END_IF
			IF ftrigAnyTablesMotorsMoving.Q OR (config_bNoHardwareTestMode AND tTimeInState>T#0.25S) THEN
				IF cmd_bReverseDirectionForWideDoor THEN
					machineState := DOOR_DASHER_CROSS_TRANSFER_RESTART_TARGET_MOTOR;
				ELSE
					machineState := DOOR_DASHER_CROSS_TRANSFER_DEACTIVATE_CROSS_CYLS;
				END_IF
			END_IF
		END_IF

	DOOR_DASHER_CROSS_TRANSFER_RESTART_TARGET_MOTOR:
        IF bFirstPass THEN
			IF bMovingFwd THEN
				targetCrossRev(); // reverse direction to find rising edge of fence-stop eye.
			ELSE
				targetCrossFwd(); // reverse direction to find falling edge of fence-stop eye.
			END_IF
			targetCrossSlower();
			rtrigTargetMotorMoving(CLK:=FALSE);
			rtrigTargetFenceEye(CLK:=FALSE);
			tonCrossFeedTargetFenceEyeValidTimer(IN:=FALSE, PT:=config_tCrossFeedTargetEyeValidTime);
		ELSE
			rtrigTargetMotorMoving(CLK:=isTargetMotorMoving());
			IF rtrigTargetMotorMoving.Q OR (config_bNoHardwareTestMode AND tTimeInState>T#0.25S) THEN
				machineState := DOOR_DASHER_CROSS_TRANSFER_FIND_RISING_EDGE_OF_TARGET_FENCE_EYE;
			END_IF
		END_IF
	
	DOOR_DASHER_CROSS_TRANSFER_FIND_RISING_EDGE_OF_TARGET_FENCE_EYE:
		IF bFirstPass THEN
			rtrigCrossTargetFenceStopEye(CLK:=FALSE);
			tonCrossFeedTargetFenceEyeValidTimer(IN:=FALSE, PT:=config_tCrossFeedTargetFenceStopEyeValidTime);
		ELSE
			tonCrossFeedTargetFenceEyeValidTimer(IN:=pdi_targetFenceStopEye^);
			rtrigCrossTargetFenceStopEye(CLK:=tonCrossFeedTargetFenceEyeValidTimer.Q);
			IF rtrigCrossTargetFenceStopEye.Q OR (config_bNoHardwareTestMode AND tTimeInState>T#0.25S) THEN
				machineState := DOOR_DASHER_CROSS_TRANSFER_STOP_MOTORS_ON_TARGET_FENCE_EYE;
			END_IF
		END_IF
	
	DOOR_DASHER_CROSS_TRANSFER_STOP_MOTORS_ON_TARGET_FENCE_EYE:
		IF bFirstPass THEN
			targetStop();
			ftrigTargetMotorMoving(CLK:=FALSE);
		ELSE
			ftrigTargetMotorMoving(CLK:=isTargetMotorMoving());
			IF ftrigTargetMotorMoving.Q OR (config_bNoHardwareTestMode AND tTimeInState>T#0.25S) THEN
				bTargetTransferTableCandDsideDoorFeedEyesClear := 
					config_bNoHardwareTestMode OR 
					isTargetTransferTableCandDsideDoorFeedEyesClear();
				IF bTargetTransferTableCandDsideDoorFeedEyesClear THEN
					machineState := DOOR_DASHER_CROSS_TRANSFER_DEACTIVATE_CROSS_CYLS;
				ELSE
					iErrorId := DOOR_DASHER_TARGET_TRANSFER_TABLE_C_AND_D_FEED_EYES_MUST_BE_CLEAR;
				END_IF
			END_IF
		END_IF
		
	DOOR_DASHER_CROSS_TRANSFER_DEACTIVATE_CROSS_CYLS:
        IF bFirstPass THEN
			deactivateTablesCrossCyls();
			bAllCrossCylsRetracted := FALSE;
		ELSE
			bAnyTableBusy := anyTableBusy();
			bAllCrossCylsRetracted := 
				allTablesCrossCylsRetracted() AND 
				NOT bAnyTableBusy AND 
				cmd_bNext;
			IF bAllCrossCylsRetracted OR (config_bNoHardwareTestMode AND tTimeInState>T#0.25S) THEN
				IF NOT bIsConveyorAtTarget THEN
					machineState := DOOR_DASHER_CROSS_TRANSFER_ALIGN_DOOR_AT_TARGET;
				ELSE
					machineState := DOOR_DASHER_CROSS_TRANSFER_WAIT_FOR_ALL_DOORDASHERS_COMPLETE;
				END_IF
			END_IF
		END_IF
	
	DOOR_DASHER_CROSS_TRANSFER_ALIGN_DOOR_AT_TARGET:
        IF bFirstPass THEN
			alignDoorAtTarget();
		ELSE
			bAligningDoorStarted:=isAligningDoorAtTarget();
			IF bAligningDoorStarted OR (config_bNoHardwareTestMode AND tTimeInState>T#0.25S) THEN
				machineState := DOOR_DASHER_CROSS_TRANSFER_WAIT_FOR_ALIGN_DOOR_AT_TARGET_COMPLETE;
			END_IF
		END_IF
		
	DOOR_DASHER_CROSS_TRANSFER_WAIT_FOR_ALIGN_DOOR_AT_TARGET_COMPLETE:
		IF bFirstPass THEN
			;
		ELSE
			bAligningDoorComplete := isAligningDoorAtTargetComplete();
			IF bAligningDoorComplete THEN
				machineState := DOOR_DASHER_CROSS_TRANSFER_WAIT_FOR_ALL_DOORDASHERS_COMPLETE;
			END_IF
		END_IF		

	DOOR_DASHER_CROSS_TRANSFER_WAIT_FOR_ALL_DOORDASHERS_COMPLETE:
		IF bFirstPass THEN
			rtrigSourceLeadingAndTrailingNeighborsComplete(CLK:=FALSE);
			bCrossTransferSourceTrailingNeighborComplete := FALSE;
			bCrossTransferSourceLeadingNeighborComplete := FALSE;
		ELSE
			IF NOT bCrossTransferSourceTrailingNeighborComplete THEN
				bCrossTransferSourceTrailingNeighborComplete := isSourceTrailingNeighborComplete();
			END_IF
			IF NOT bCrossTransferSourceLeadingNeighborComplete THEN
				bCrossTransferSourceLeadingNeighborComplete := isSourceLeadingNeighborComplete();
			END_IF
			bAnyTableBusy := anyTableBusy();
			rtrigSourceLeadingAndTrailingNeighborsComplete(CLK:=
				cmd_bNext AND
				NOT bAnyTableBusy AND
				bCrossTransferSourceLeadingNeighborComplete AND 
				bCrossTransferSourceTrailingNeighborComplete);
			IF rtrigSourceLeadingAndTrailingNeighborsComplete.CLK THEN
				machineState := DOOR_DASHER_CROSS_TRANSFER_COMPLETE;
			END_IF
		END_IF
		
	DOOR_DASHER_CROSS_TRANSFER_COMPLETE:
        IF bFirstPass THEN	
			bCrossTransferSeqRunning	:= FALSE;
		ELSIF cmd_bNext THEN
			machineState := DOOR_DASHER_SET_SOURCE_AND_TARGET_INTERNAL;
		END_IF

	DOOR_DASHER_INLINE_TRANSFER_START:
		IF bFirstPass THEN
			inlineTransferStart();
			bInlineTransferSeqRunning	:= TRUE;
			bAllSourceAndTargetExternal := FALSE;
			bAllCrossCylsRetracted := FALSE;
		ELSE
			IF cmd_bNext THEN
				machineState := DOOR_DASHER_INLINE_TRANSFER_DEACTIVATE_CROSS_CYLS;	
			END_IF
		END_IF
		
	DOOR_DASHER_INLINE_TRANSFER_DEACTIVATE_CROSS_CYLS:
		IF bFirstPass THEN
			deactivateTablesCrossCyls();
			bAllCrossCylsRetracted := FALSE;
		ELSE
			bAnyTableBusy := anyTableBusy();
			bAllCrossCylsRetracted := allTablesCrossCylsRetracted() AND 
				NOT bAnyTableBusy AND 
				tTimeInState>T#20MS AND // don't know why have to wait for at least 20ms to start motor. 
				cmd_bNext;
			IF bAllCrossCylsRetracted OR (config_bNoHardwareTestMode AND tTimeInState>T#0.25S) THEN
				IF pdi_inlineSourceFeedEyeRisingEdge^ THEN
					machineState := DOOR_DASHER_INLINE_TRANSFER_WAIT_FOR_ALL_DOORDASHERS_READY;
				ELSE
					machineState := DOOR_DASHER_INLINE_TRANSFER_START_SOURCE_MOTOR;
				END_IF
			END_IF	
		END_IF
		
	DOOR_DASHER_INLINE_TRANSFER_START_SOURCE_MOTOR:
		IF bFirstPass THEN
			IF bMovingFwd THEN
				sourceGoFwd();
			ELSE
				sourceGoRev();
			END_IF
			sourceGoFast();
			rtrigSourceMotorMoving(CLK:=FALSE);
		ELSE
			rtrigSourceMotorMoving(CLK:=isSourceMotorMoving());
			IF rtrigSourceMotorMoving.Q OR (config_bNoHardwareTestMode AND tTimeInState>T#0.25S) THEN
				machineState := DOOR_DASHER_INLINE_TRANSFER_FIND_SOURCE_EYE_RISING_EDGE;
			END_IF
		END_IF
		
		
	DOOR_DASHER_INLINE_TRANSFER_FIND_SOURCE_EYE_RISING_EDGE:
		IF bFirstPass THEN
			rtrigInlineSourceFeedEye(CLK:=FALSE);
			tonInlineFeedSourceEyeValidTimer(IN:=FALSE, PT:=config_tInlineFeedSourceEyeValidTime);
		ELSE
			tonInlineFeedSourceEyeValidTimer(IN:=pdi_inlineSourceFeedEyeRisingEdge^);
			rtrigInlineSourceFeedEye(CLK:=tonInlineFeedSourceEyeValidTimer.Q);
			IF rtrigInlineSourceFeedEye.Q OR (config_bNoHardwareTestMode AND tTimeInState>T#0.25S) THEN
				machineState := DOOR_DASHER_INLINE_TRANSFER_STOP_SOURCE_MOTOR;
			ELSIF tTimeInState > config_tFindSourceInlineEyeMaxTimeSec THEN
				IF bMovingFwd THEN
					iErrorId := DOOR_DASHER_FAILED_TO_FIND_SOURCE_B_EYE_RISING_EDGE;
				ELSE
					iErrorId := DOOR_DASHER_FAILED_TO_FIND_SOURCE_A_EYE_RISING_EDGE;
				END_IF
			END_IF
		END_IF
		
	DOOR_DASHER_INLINE_TRANSFER_STOP_SOURCE_MOTOR:
		IF bFirstPass THEN
			sourceStop();
			ftrigSourceMotorMoving(CLK:=FALSE);
		ELSE
			ftrigSourceMotorMoving(CLK:=isSourceMotorMoving());
			IF ftrigSourceMotorMoving.Q OR (config_bNoHardwareTestMode AND tTimeInState>T#0.25S) THEN
				machineState := DOOR_DASHER_INLINE_TRANSFER_WAIT_FOR_ALL_DOORDASHERS_READY;
			END_IF
		END_IF
		
	DOOR_DASHER_INLINE_TRANSFER_WAIT_FOR_ALL_DOORDASHERS_READY:
		IF bFirstPass THEN
			rtrigSourceLeadingAndTrailingNeighborsReady(CLK:=FALSE);
			bInlineTransferSourceTrailingNeighborReady := FALSE;
			bInlineTransferSourceLeadingNeighborReady := FALSE;
		ELSE
			IF NOT bInlineTransferSourceTrailingNeighborReady THEN
				bInlineTransferSourceTrailingNeighborReady := isSourceTrailingNeighborReady();
			END_IF
			IF NOT bInlineTransferSourceLeadingNeighborReady THEN
				bInlineTransferSourceLeadingNeighborReady := isSourceLeadingNeighborReady();
			END_IF
			rtrigSourceLeadingAndTrailingNeighborsReady(CLK:=
				cmd_bNext AND
				bInlineTransferSourceLeadingNeighborReady AND 
				bInlineTransferSourceTrailingNeighborReady
				);
			IF rtrigSourceLeadingAndTrailingNeighborsReady.Q THEN
				machineState := DOOR_DASHER_INLINE_TRANSFER_START_MOTORS;
			END_IF
		END_IF
		
	DOOR_DASHER_INLINE_TRANSFER_START_MOTORS:
		IF bFirstPass THEN
			IF bMovingFwd THEN
				goFwd();
			ELSE
				goRev();
			END_IF
			goFast();
			rtrigAllTablesMotorsMoving(CLK:=FALSE);
		ELSE
			rtrigAllTablesMotorsMoving(CLK:=allTablesMotorsMoving());
			IF rtrigAllTablesMotorsMoving.Q OR (config_bNoHardwareTestMode AND tTimeInState>T#5.25S) THEN
				machineState := DOOR_DASHER_INLINE_TRANSFER_FIND_TARGET_EYE_RISING_EDGE;
			END_IF
		END_IF
		
	DOOR_DASHER_INLINE_TRANSFER_FIND_TARGET_EYE_RISING_EDGE:
		IF bFirstPass THEN
			rtrigInlineTargetFeedEyeRising(CLK:=FALSE);
			tonInlineFeedTargetEyeRisingValidTimer(IN:=FALSE, PT:=config_tInlineFeedTargetEyeRisingValidTime);
		ELSE
			tonInlineFeedTargetEyeRisingValidTimer(IN:=pdi_inlineTargetFeedEyeRisingEdge^);
			rtrigInlineTargetFeedEyeRising(CLK:=tonInlineFeedTargetEyeRisingValidTimer.Q);
			IF rtrigInlineTargetFeedEyeRising.Q OR (config_bNoHardwareTestMode AND tTimeInState>T#0.25S) THEN
				machineState := DOOR_DASHER_INLINE_TRANSFER_FIND_TARGET_EYE_FALLING_EDGE;
			ELSIF tTimeInState > config_tInlineFeedTargetEyeRisingMaxTime THEN
				IF bMovingFwd THEN
					iErrorId := DOOR_DASHER_FAILED_TO_FIND_TARGET_A_SIDE_EYE_RISING;
				ELSE
					iErrorId := DOOR_DASHER_FAILED_TO_FIND_TARGET_B_SIDE_EYE_RISING;
				END_IF
			END_IF
		END_IF
		
	DOOR_DASHER_INLINE_TRANSFER_FIND_TARGET_EYE_FALLING_EDGE:
		IF bFirstPass THEN
			ftrigInlineTargetFeedEyeFalling(CLK:=FALSE);
			tofInlineTargetFeedEyeFallingEdgeTimer(IN:=FALSE, PT:=config_tInlineTargetFeedEyeFallingEdgeTime);
		ELSE
			tofInlineTargetFeedEyeFallingEdgeTimer(IN:=pdi_inlineTargetFeedEyeFallingEdge^);
			ftrigInlineTargetFeedEyeFalling(CLK:=tofInlineTargetFeedEyeFallingEdgeTimer.Q);
			IF ftrigInlineTargetFeedEyeFalling.Q OR (config_bNoHardwareTestMode AND tTimeInState>T#0.25S) THEN
				machineState := DOOR_DASHER_INLINE_TRANSFER_STOP_MOTORS;
			ELSIF tTimeInState > config_tInlineFeedTargetEyeFallingMaxTime THEN
				IF bMovingFwd THEN
					iErrorId := DOOR_DASHER_FAILED_TO_FIND_TARGET_A_SIDE_EYE_FALLING;
				ELSE
					iErrorId := DOOR_DASHER_FAILED_TO_FIND_TARGET_B_SIDE_EYE_FALLING;
				END_IF
			END_IF
		END_IF
		
	DOOR_DASHER_INLINE_TRANSFER_STOP_MOTORS:
		IF bFirstPass THEN
			stop();
			ftrigAnyTablesMotorsMoving(CLK:=FALSE);
			tofStopMotorValidTimer(IN:=FALSE, PT:=config_tStopMotorValidTime);
		ELSE
			tofStopMotorValidTimer(IN:=anyTableMotorMoving());
			ftrigAnyTablesMotorsMoving(CLK:=tofStopMotorValidTimer.Q);
			
			IF ftrigAnyTablesMotorsMoving.Q OR (config_bNoHardwareTestMode AND tTimeInState>T#0.25S) THEN
				IF bIsTargetBufferTable THEN
					machineState := DOOR_DASHER_INLINE_TRANSFER_WAIT_FOR_ALL_DOORDASHERS_COMPLETE;
				ELSE	
					machineState := DOOR_DASHER_INLINE_TRANSFER_FEEDIN_DOOR_AT_TARGET;
				END_IF

			END_IF
		END_IF
		
	DOOR_DASHER_INLINE_TRANSFER_FEEDIN_DOOR_AT_TARGET:
		IF bFirstPass THEN
			feedinDoorAtTarget();
		ELSE
			bFeedingInDoorStarted:=isFeedingInDoorAtTarget();
			IF bFeedingInDoorStarted THEN
				machineState := DOOR_DASHER_INLINE_TRANSFER_WAIT_FOR_FEEDIN_DOOR_AT_TARGET_COMPLETE;
			END_IF
		END_IF
		
	DOOR_DASHER_INLINE_TRANSFER_WAIT_FOR_FEEDIN_DOOR_AT_TARGET_COMPLETE:
		IF bFirstPass THEN
			;
		ELSE
			bFeedingInDoorComplete := isFeedingInDoorAtTargetComplete();
			IF bFeedingInDoorComplete THEN
				machineState := DOOR_DASHER_INLINE_TRANSFER_WAIT_FOR_ALL_DOORDASHERS_COMPLETE;
			END_IF
		END_IF		
		
	DOOR_DASHER_INLINE_TRANSFER_WAIT_FOR_ALL_DOORDASHERS_COMPLETE:
		IF bFirstPass THEN
			rtrigSourceLeadingAndTrailingNeighborsComplete(CLK:=FALSE);
			bInlineTransferSourceTrailingNeighborComplete := FALSE;
			bInlineTransferSourceLeadingNeighborComplete := FALSE;
		ELSE
			IF NOT bInlineTransferSourceTrailingNeighborComplete THEN
				bInlineTransferSourceTrailingNeighborComplete := isSourceTrailingNeighborComplete();
			END_IF
			IF NOT bInlineTransferSourceLeadingNeighborComplete THEN
				bInlineTransferSourceLeadingNeighborComplete := isSourceLeadingNeighborComplete();
			END_IF
			bAnyTableBusy := anyTableBusy();
			rtrigSourceLeadingAndTrailingNeighborsComplete(CLK:=
				cmd_bNext AND
				NOT bAnyTableBusy AND
				bInlineTransferSourceLeadingNeighborComplete AND 
				bInlineTransferSourceTrailingNeighborComplete);
			IF rtrigSourceLeadingAndTrailingNeighborsComplete.CLK THEN
				machineState := DOOR_DASHER_INLINE_TRANSFER_COMPLETE;
			END_IF
		END_IF
	
	DOOR_DASHER_INLINE_TRANSFER_COMPLETE:
		IF bFirstPass THEN
			bInlineTransferSeqRunning	:= FALSE;
		ELSIF cmd_bNext THEN
			machineState := DOOR_DASHER_SET_SOURCE_AND_TARGET_INTERNAL;
		END_IF
	
	DOOR_DASHER_SET_SOURCE_AND_TARGET_INTERNAL:
        IF bFirstPass THEN
			setInternal();
		END_IF
		bAnyTableExternal := anyTableExternal();
        IF NOT bAnyTableExternal THEN
			machineState := DOOR_DASHER_COMPLETE;
		END_IF
		
	DOOR_DASHER_COMPLETE:
		IF bFirstPass THEN
			status_bBusy := FALSE;
			IF bTransferring THEN
				bTransferring := FALSE;
				updateSourceTargetDoorTrack();
				setTargetDoorTransferredInCompleted();
			END_IF
		ELSIF cmd_bNext THEN
			machineState := DOOR_DASHER_AUTOFEED_ON;
		END_IF
		
	DOOR_DASHER_ERROR:
		IF bFirstPass THEN
			status_bBusy := FALSE;
			status_bReady := FALSE;
			bError := TRUE;
			stop();
		END_IF
		IF NOT cmd_bEnable THEN
			machineState := DOOR_DASHER_DISABLED;
		ELSIF cmd_bReset THEN
			clearLastError();
			machineState := DOOR_DASHER_AUTOFEED_OFF;
		END_IF


END_CASE
END_METHOD

(* The UML-statechart version of the Structured-Text version of doState method.  
	The derived function block of KvalStateMachineBase_UmlSC should override/extend this method.  *)
METHOD doState_UmlSC
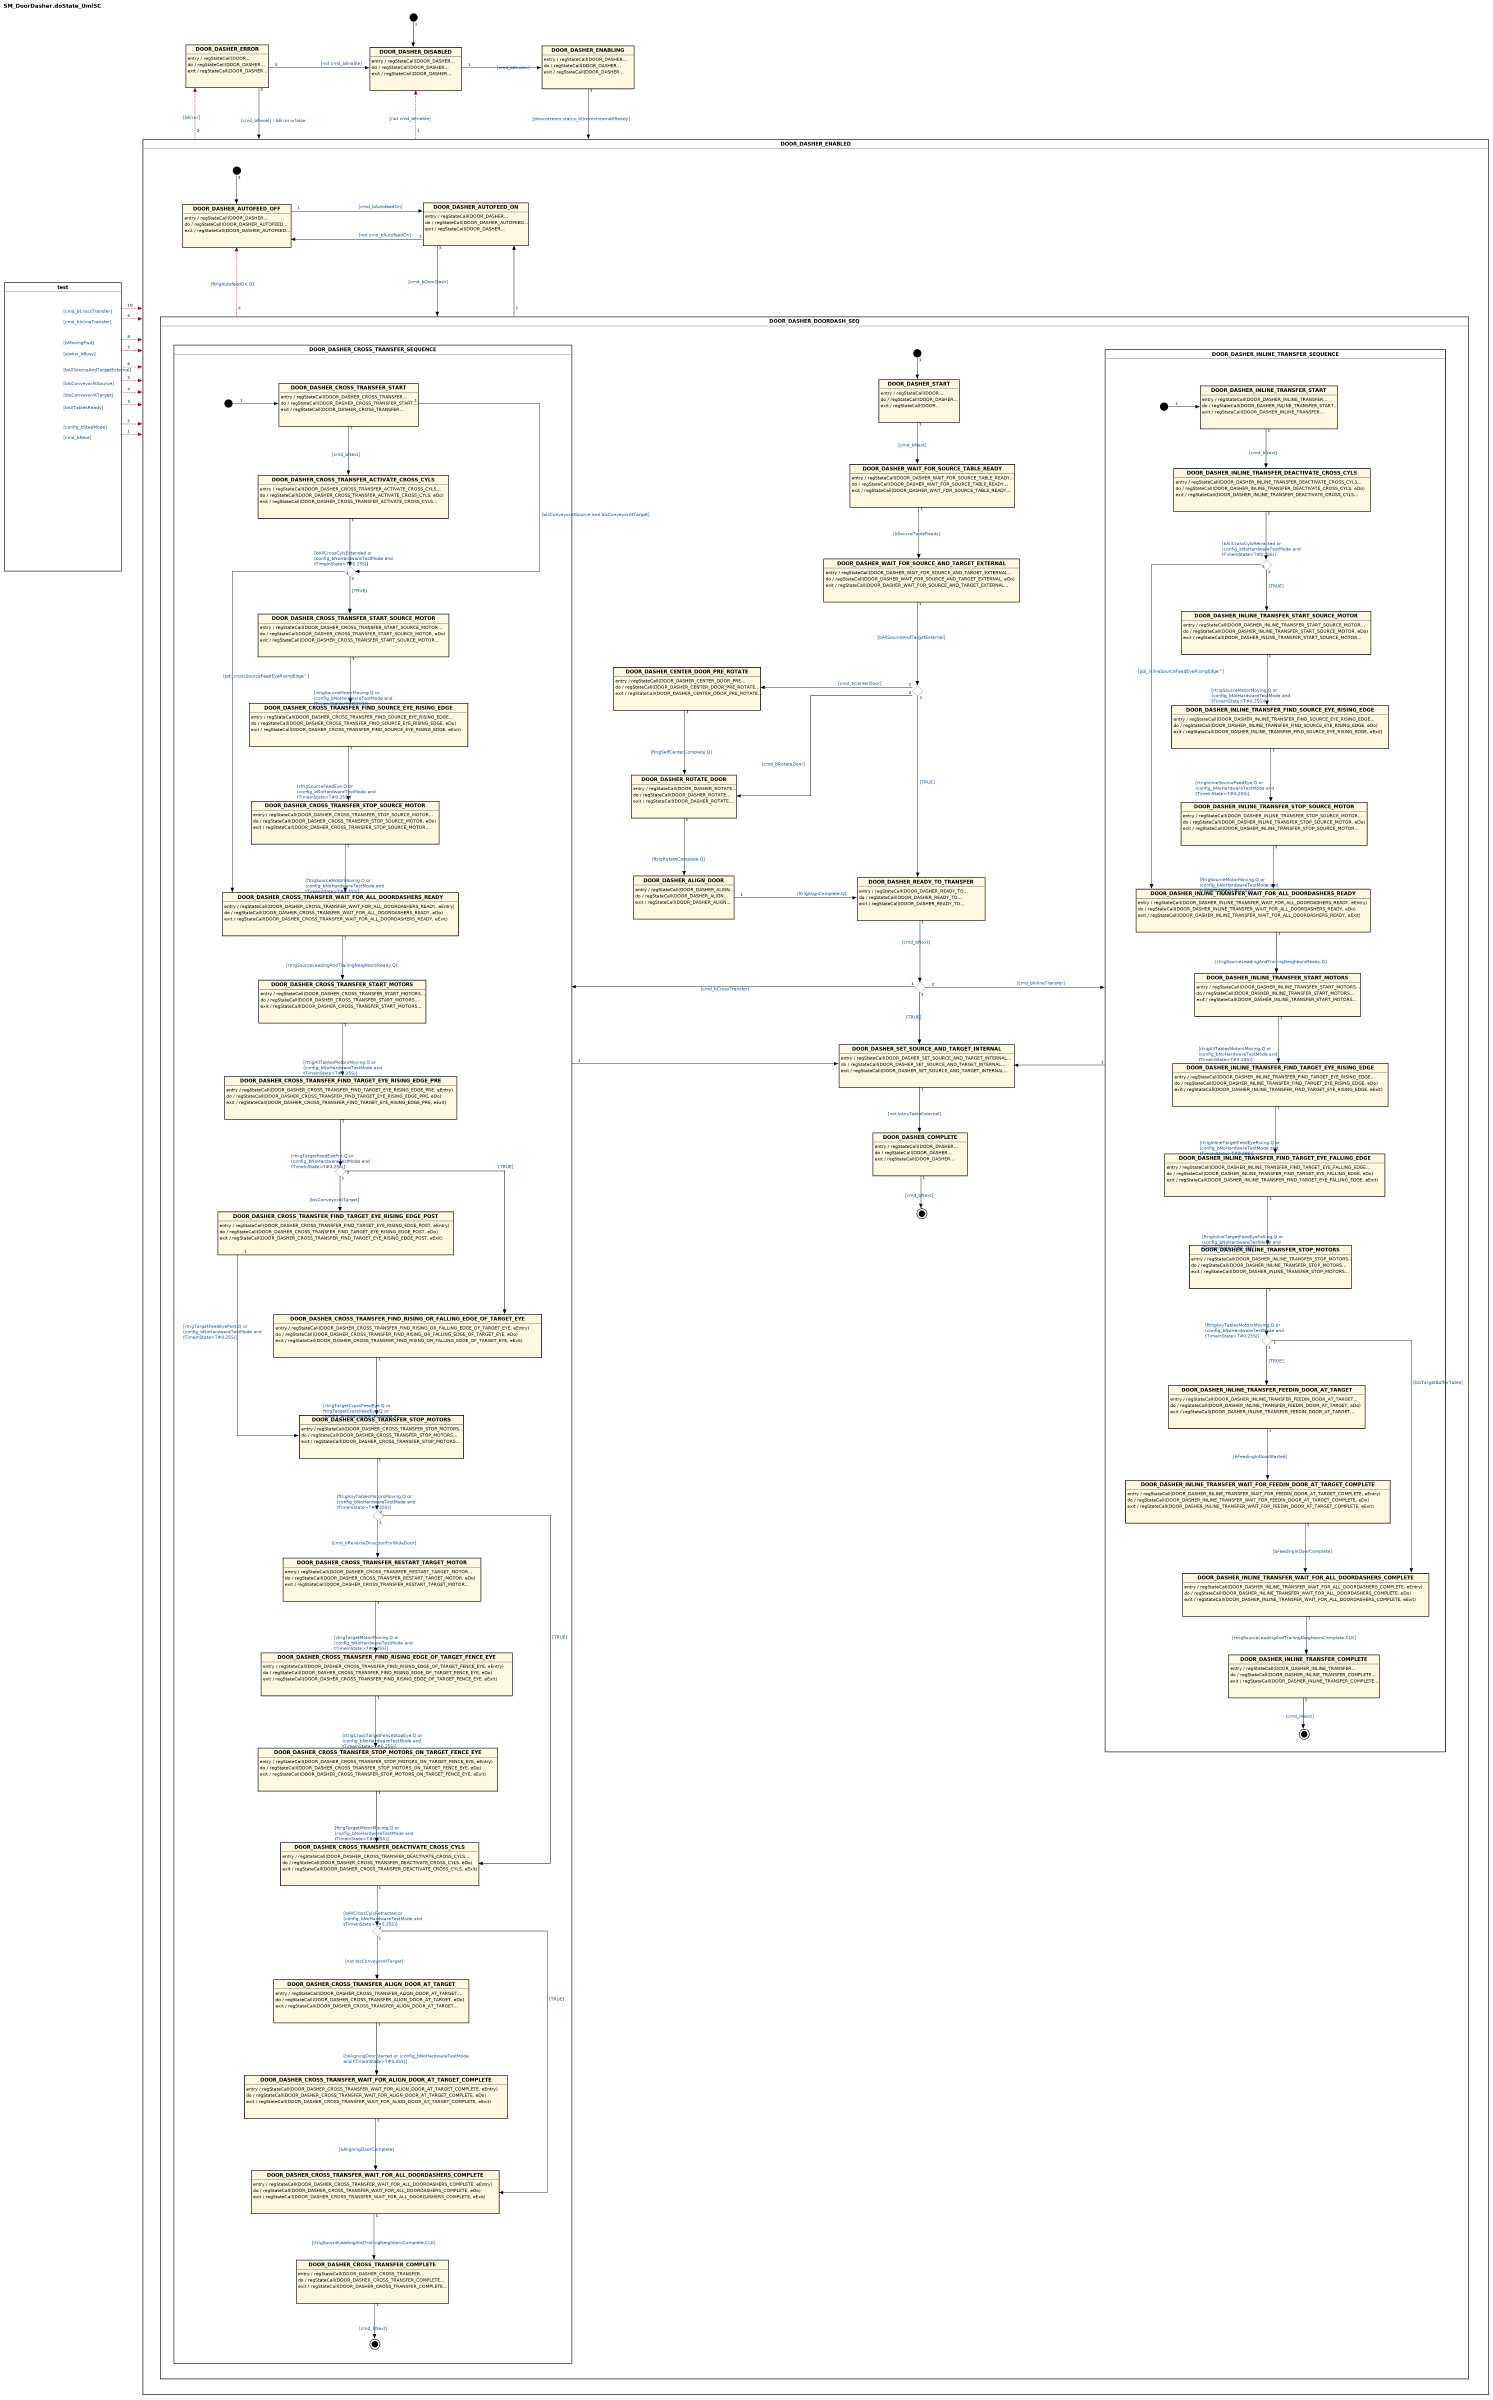
STATECHART doState_UmlSC  // abortable
    START StartState1
    STATE DOOR_DASHER_ERROR
        entry / regStateCall(DOOR_DASHER_ERROR, eEntry)
        do / regStateCall(DOOR_DASHER_ERROR, eDo)
        exit / regStateCall(DOOR_DASHER_ERROR, eExit)
    STATE DOOR_DASHER_DISABLED
        entry / regStateCall(DOOR_DASHER_DISABLED, eEntry)
        do / regStateCall(DOOR_DASHER_DISABLED, eDo)
        exit / regStateCall(DOOR_DASHER_DISABLED, eExit)
    STATE DOOR_DASHER_ENABLING
        entry / regStateCall(DOOR_DASHER_ENABLING, eEntry)
        do / regStateCall(DOOR_DASHER_ENABLING, eDo)
        exit / regStateCall(DOOR_DASHER_ENABLING, eExit)
    COMPOSITE STATE DOOR_DASHER_ENABLED
        START StartState2
        STATE DOOR_DASHER_AUTOFEED_OFF
            entry / regStateCall(DOOR_DASHER_AUTOFEED_OFF, eEntry)
            do / regStateCall(DOOR_DASHER_AUTOFEED_OFF, eDo)
            exit / regStateCall(DOOR_DASHER_AUTOFEED_OFF, eExit)
        STATE DOOR_DASHER_AUTOFEED_ON
            entry / regStateCall(DOOR_DASHER_AUTOFEED_ON, eEntry)
            do / regStateCall(DOOR_DASHER_AUTOFEED_ON, eDo)
            exit / regStateCall(DOOR_DASHER_AUTOFEED_ON, eExit)
        COMPOSITE STATE DOOR_DASHER_DOORDASH_SEQ
            START StartState4
            COMPOSITE STATE DOOR_DASHER_CROSS_TRANSFER_SEQUENCE
                START StartState3
                STATE DOOR_DASHER_CROSS_TRANSFER_START
                    entry / regStateCall(DOOR_DASHER_CROSS_TRANSFER_START, eEntry)
                    do / regStateCall(DOOR_DASHER_CROSS_TRANSFER_START, eDo)
                    exit / regStateCall(DOOR_DASHER_CROSS_TRANSFER_START, eExit)
                STATE DOOR_DASHER_CROSS_TRANSFER_ACTIVATE_CROSS_CYLS
                    entry / regStateCall(DOOR_DASHER_CROSS_TRANSFER_ACTIVATE_CROSS_CYLS, eEntry)
                    do / regStateCall(DOOR_DASHER_CROSS_TRANSFER_ACTIVATE_CROSS_CYLS, eDo)
                    exit / regStateCall(DOOR_DASHER_CROSS_TRANSFER_ACTIVATE_CROSS_CYLS, eExit)
                CHOICE ChoiceElement6
                STATE DOOR_DASHER_CROSS_TRANSFER_START_SOURCE_MOTOR
                    entry / regStateCall(DOOR_DASHER_CROSS_TRANSFER_START_SOURCE_MOTOR, eEntry)
                    do / regStateCall(DOOR_DASHER_CROSS_TRANSFER_START_SOURCE_MOTOR, eDo)
                    exit / regStateCall(DOOR_DASHER_CROSS_TRANSFER_START_SOURCE_MOTOR, eExit)
                STATE DOOR_DASHER_CROSS_TRANSFER_FIND_SOURCE_EYE_RISING_EDGE
                    entry / regStateCall(DOOR_DASHER_CROSS_TRANSFER_FIND_SOURCE_EYE_RISING_EDGE, eEntry)
                    do / regStateCall(DOOR_DASHER_CROSS_TRANSFER_FIND_SOURCE_EYE_RISING_EDGE, eDo)
                    exit / regStateCall(DOOR_DASHER_CROSS_TRANSFER_FIND_SOURCE_EYE_RISING_EDGE, eExit)
                STATE DOOR_DASHER_CROSS_TRANSFER_STOP_SOURCE_MOTOR
                    entry / regStateCall(DOOR_DASHER_CROSS_TRANSFER_STOP_SOURCE_MOTOR, eEntry)
                    do / regStateCall(DOOR_DASHER_CROSS_TRANSFER_STOP_SOURCE_MOTOR, eDo)
                    exit / regStateCall(DOOR_DASHER_CROSS_TRANSFER_STOP_SOURCE_MOTOR, eExit)
                STATE DOOR_DASHER_CROSS_TRANSFER_WAIT_FOR_ALL_DOORDASHERS_READY
                    entry / regStateCall(DOOR_DASHER_CROSS_TRANSFER_WAIT_FOR_ALL_DOORDASHERS_READY, eEntry)
                    do / regStateCall(DOOR_DASHER_CROSS_TRANSFER_WAIT_FOR_ALL_DOORDASHERS_READY, eDo)
                    exit / regStateCall(DOOR_DASHER_CROSS_TRANSFER_WAIT_FOR_ALL_DOORDASHERS_READY, eExit)
                STATE DOOR_DASHER_CROSS_TRANSFER_START_MOTORS
                    entry / regStateCall(DOOR_DASHER_CROSS_TRANSFER_START_MOTORS, eEntry)
                    do / regStateCall(DOOR_DASHER_CROSS_TRANSFER_START_MOTORS, eDo)
                    exit / regStateCall(DOOR_DASHER_CROSS_TRANSFER_START_MOTORS, eExit)
                STATE DOOR_DASHER_CROSS_TRANSFER_FIND_TARGET_EYE_RISING_EDGE_PRE
                    entry / regStateCall(DOOR_DASHER_CROSS_TRANSFER_FIND_TARGET_EYE_RISING_EDGE_PRE, eEntry)
                    do / regStateCall(DOOR_DASHER_CROSS_TRANSFER_FIND_TARGET_EYE_RISING_EDGE_PRE, eDo)
                    exit / regStateCall(DOOR_DASHER_CROSS_TRANSFER_FIND_TARGET_EYE_RISING_EDGE_PRE, eExit)
                CHOICE ChoiceElement3
                STATE DOOR_DASHER_CROSS_TRANSFER_FIND_TARGET_EYE_RISING_EDGE_POST
                    entry / regStateCall(DOOR_DASHER_CROSS_TRANSFER_FIND_TARGET_EYE_RISING_EDGE_POST, eEntry)
                    do / regStateCall(DOOR_DASHER_CROSS_TRANSFER_FIND_TARGET_EYE_RISING_EDGE_POST, eDo)
                    exit / regStateCall(DOOR_DASHER_CROSS_TRANSFER_FIND_TARGET_EYE_RISING_EDGE_POST, eExit)
                STATE DOOR_DASHER_CROSS_TRANSFER_FIND_RISING_OR_FALLING_EDGE_OF_TARGET_EYE
                    entry / regStateCall(DOOR_DASHER_CROSS_TRANSFER_FIND_RISING_OR_FALLING_EDGE_OF_TARGET_EYE, eEntry)
                    do / regStateCall(DOOR_DASHER_CROSS_TRANSFER_FIND_RISING_OR_FALLING_EDGE_OF_TARGET_EYE, eDo)
                    exit / regStateCall(DOOR_DASHER_CROSS_TRANSFER_FIND_RISING_OR_FALLING_EDGE_OF_TARGET_EYE, eExit)
                STATE DOOR_DASHER_CROSS_TRANSFER_STOP_MOTORS
                    entry / regStateCall(DOOR_DASHER_CROSS_TRANSFER_STOP_MOTORS, eEntry)
                    do / regStateCall(DOOR_DASHER_CROSS_TRANSFER_STOP_MOTORS, eDo)
                    exit / regStateCall(DOOR_DASHER_CROSS_TRANSFER_STOP_MOTORS, eExit)
                CHOICE ChoiceElement2
                STATE DOOR_DASHER_CROSS_TRANSFER_RESTART_TARGET_MOTOR
                    entry / regStateCall(DOOR_DASHER_CROSS_TRANSFER_RESTART_TARGET_MOTOR, eEntry)
                    do / regStateCall(DOOR_DASHER_CROSS_TRANSFER_RESTART_TARGET_MOTOR, eDo)
                    exit / regStateCall(DOOR_DASHER_CROSS_TRANSFER_RESTART_TARGET_MOTOR, eExit)
                STATE DOOR_DASHER_CROSS_TRANSFER_FIND_RISING_EDGE_OF_TARGET_FENCE_EYE
                    entry / regStateCall(DOOR_DASHER_CROSS_TRANSFER_FIND_RISING_EDGE_OF_TARGET_FENCE_EYE, eEntry)
                    do / regStateCall(DOOR_DASHER_CROSS_TRANSFER_FIND_RISING_EDGE_OF_TARGET_FENCE_EYE, eDo)
                    exit / regStateCall(DOOR_DASHER_CROSS_TRANSFER_FIND_RISING_EDGE_OF_TARGET_FENCE_EYE, eExit)
                STATE DOOR_DASHER_CROSS_TRANSFER_STOP_MOTORS_ON_TARGET_FENCE_EYE
                    entry / regStateCall(DOOR_DASHER_CROSS_TRANSFER_STOP_MOTORS_ON_TARGET_FENCE_EYE, eEntry)
                    do / regStateCall(DOOR_DASHER_CROSS_TRANSFER_STOP_MOTORS_ON_TARGET_FENCE_EYE, eDo)
                    exit / regStateCall(DOOR_DASHER_CROSS_TRANSFER_STOP_MOTORS_ON_TARGET_FENCE_EYE, eExit)
                STATE DOOR_DASHER_CROSS_TRANSFER_DEACTIVATE_CROSS_CYLS
                    entry / regStateCall(DOOR_DASHER_CROSS_TRANSFER_DEACTIVATE_CROSS_CYLS, eEntry)
                    do / regStateCall(DOOR_DASHER_CROSS_TRANSFER_DEACTIVATE_CROSS_CYLS, eDo)
                    exit / regStateCall(DOOR_DASHER_CROSS_TRANSFER_DEACTIVATE_CROSS_CYLS, eExit)
                CHOICE ChoiceElement1
                STATE DOOR_DASHER_CROSS_TRANSFER_ALIGN_DOOR_AT_TARGET
                    entry / regStateCall(DOOR_DASHER_CROSS_TRANSFER_ALIGN_DOOR_AT_TARGET, eEntry)
                    do / regStateCall(DOOR_DASHER_CROSS_TRANSFER_ALIGN_DOOR_AT_TARGET, eDo)
                    exit / regStateCall(DOOR_DASHER_CROSS_TRANSFER_ALIGN_DOOR_AT_TARGET, eExit)
                STATE DOOR_DASHER_CROSS_TRANSFER_WAIT_FOR_ALIGN_DOOR_AT_TARGET_COMPLETE
                    entry / regStateCall(DOOR_DASHER_CROSS_TRANSFER_WAIT_FOR_ALIGN_DOOR_AT_TARGET_COMPLETE, eEntry)
                    do / regStateCall(DOOR_DASHER_CROSS_TRANSFER_WAIT_FOR_ALIGN_DOOR_AT_TARGET_COMPLETE, eDo)
                    exit / regStateCall(DOOR_DASHER_CROSS_TRANSFER_WAIT_FOR_ALIGN_DOOR_AT_TARGET_COMPLETE, eExit)
                STATE DOOR_DASHER_CROSS_TRANSFER_WAIT_FOR_ALL_DOORDASHERS_COMPLETE
                    entry / regStateCall(DOOR_DASHER_CROSS_TRANSFER_WAIT_FOR_ALL_DOORDASHERS_COMPLETE, eEntry)
                    do / regStateCall(DOOR_DASHER_CROSS_TRANSFER_WAIT_FOR_ALL_DOORDASHERS_COMPLETE, eDo)
                    exit / regStateCall(DOOR_DASHER_CROSS_TRANSFER_WAIT_FOR_ALL_DOORDASHERS_COMPLETE, eExit)
                STATE DOOR_DASHER_CROSS_TRANSFER_COMPLETE
                    entry / regStateCall(DOOR_DASHER_CROSS_TRANSFER_COMPLETE, eEntry)
                    do / regStateCall(DOOR_DASHER_CROSS_TRANSFER_COMPLETE, eDo)
                    exit / regStateCall(DOOR_DASHER_CROSS_TRANSFER_COMPLETE, eExit)
                END EndState1
                StartState3 -> DOOR_DASHER_CROSS_TRANSFER_START  // priority 1, on completion
                DOOR_DASHER_CROSS_TRANSFER_START -> ChoiceElement6 [bIsConveyorAtSource and bIsConveyorAtTarget] // priority 1
                DOOR_DASHER_CROSS_TRANSFER_START -> DOOR_DASHER_CROSS_TRANSFER_ACTIVATE_CROSS_CYLS [cmd_bNext] // priority 2
                DOOR_DASHER_CROSS_TRANSFER_ACTIVATE_CROSS_CYLS -> ChoiceElement6 [bAllCrossCylsExtended or (config_bNoHardwareTestMode and tTimeInState>T#0.25S)] // priority 1
                ChoiceElement6 -> DOOR_DASHER_CROSS_TRANSFER_WAIT_FOR_ALL_DOORDASHERS_READY [pdi_crossSourceFeedEyeRisingEdge^] // priority 1
                ChoiceElement6 -> DOOR_DASHER_CROSS_TRANSFER_START_SOURCE_MOTOR [TRUE] // priority 2
                DOOR_DASHER_CROSS_TRANSFER_START_SOURCE_MOTOR -> DOOR_DASHER_CROSS_TRANSFER_FIND_SOURCE_EYE_RISING_EDGE [rtrigSourceMotorMoving.Q or (config_bNoHardwareTestMode and tTimeInState>T#0.25S)] // priority 1, rising edge
                DOOR_DASHER_CROSS_TRANSFER_FIND_SOURCE_EYE_RISING_EDGE -> DOOR_DASHER_CROSS_TRANSFER_STOP_SOURCE_MOTOR [rtrigSourceFeedEye.Q or (config_bNoHardwareTestMode and tTimeInState>T#0.25S)] // priority 1, rising edge
                DOOR_DASHER_CROSS_TRANSFER_STOP_SOURCE_MOTOR -> DOOR_DASHER_CROSS_TRANSFER_WAIT_FOR_ALL_DOORDASHERS_READY [ftrigSourceMotorMoving.Q or (config_bNoHardwareTestMode and tTimeInState>T#0.25S)] // priority 1, rising edge
                DOOR_DASHER_CROSS_TRANSFER_WAIT_FOR_ALL_DOORDASHERS_READY -> DOOR_DASHER_CROSS_TRANSFER_START_MOTORS [rtrigSourceLeadingAndTrailingNeighborsReady.Q] // priority 1, rising edge
                DOOR_DASHER_CROSS_TRANSFER_START_MOTORS -> DOOR_DASHER_CROSS_TRANSFER_FIND_TARGET_EYE_RISING_EDGE_PRE [rtrigAllTablesMotorsMoving.Q or (config_bNoHardwareTestMode and tTimeInState>T#5.25S)] // priority 1, rising edge
                DOOR_DASHER_CROSS_TRANSFER_FIND_TARGET_EYE_RISING_EDGE_PRE -> ChoiceElement3 [rtrigTargetFeedEyePre.Q or (config_bNoHardwareTestMode and tTimeInState>T#0.25S)] // priority 1, rising edge
                ChoiceElement3 -> DOOR_DASHER_CROSS_TRANSFER_FIND_TARGET_EYE_RISING_EDGE_POST [bIsConveyorAtTarget] // priority 1
                ChoiceElement3 -> DOOR_DASHER_CROSS_TRANSFER_FIND_RISING_OR_FALLING_EDGE_OF_TARGET_EYE [TRUE] // priority 2
                DOOR_DASHER_CROSS_TRANSFER_FIND_TARGET_EYE_RISING_EDGE_POST -> DOOR_DASHER_CROSS_TRANSFER_STOP_MOTORS [rtrigTargetFeedEyePost.Q or (config_bNoHardwareTestMode and tTimeInState>T#0.25S)] // priority 1, rising edge
                DOOR_DASHER_CROSS_TRANSFER_FIND_RISING_OR_FALLING_EDGE_OF_TARGET_EYE -> DOOR_DASHER_CROSS_TRANSFER_STOP_MOTORS [rtrigTargetCrossFeedEye.Q or ftrigTargetCrossFeedEye.Q or (config_bNoHardwareTestMode and tTimeInState>T#0.25S)] // priority 1, rising edge
                DOOR_DASHER_CROSS_TRANSFER_STOP_MOTORS -> ChoiceElement2 [ftrigAnyTablesMotorsMoving.Q or (config_bNoHardwareTestMode and tTimeInState>T#0.25S)] // priority 1, rising edge
                ChoiceElement2 -> DOOR_DASHER_CROSS_TRANSFER_RESTART_TARGET_MOTOR [cmd_bReverseDirectionForWideDoor] // priority 1
                ChoiceElement2 -> DOOR_DASHER_CROSS_TRANSFER_DEACTIVATE_CROSS_CYLS [TRUE] // priority 2
                DOOR_DASHER_CROSS_TRANSFER_RESTART_TARGET_MOTOR -> DOOR_DASHER_CROSS_TRANSFER_FIND_RISING_EDGE_OF_TARGET_FENCE_EYE [rtrigTargetMotorMoving.Q or (config_bNoHardwareTestMode and tTimeInState>T#0.25S)] // priority 1, rising edge
                DOOR_DASHER_CROSS_TRANSFER_FIND_RISING_EDGE_OF_TARGET_FENCE_EYE -> DOOR_DASHER_CROSS_TRANSFER_STOP_MOTORS_ON_TARGET_FENCE_EYE [rtrigCrossTargetFenceStopEye.Q or (config_bNoHardwareTestMode and tTimeInState>T#0.25S)] // priority 1, rising edge
                DOOR_DASHER_CROSS_TRANSFER_STOP_MOTORS_ON_TARGET_FENCE_EYE -> DOOR_DASHER_CROSS_TRANSFER_DEACTIVATE_CROSS_CYLS [ftrigTargetMotorMoving.Q or (config_bNoHardwareTestMode and tTimeInState>T#0.25S)] // priority 1, rising edge
                DOOR_DASHER_CROSS_TRANSFER_DEACTIVATE_CROSS_CYLS -> ChoiceElement1 [bAllCrossCylsRetracted or (config_bNoHardwareTestMode and tTimeInState>T#0.25S)] // priority 1
                ChoiceElement1 -> DOOR_DASHER_CROSS_TRANSFER_ALIGN_DOOR_AT_TARGET [not bIsConveyorAtTarget] // priority 1
                ChoiceElement1 -> DOOR_DASHER_CROSS_TRANSFER_WAIT_FOR_ALL_DOORDASHERS_COMPLETE [TRUE] // priority 2
                DOOR_DASHER_CROSS_TRANSFER_ALIGN_DOOR_AT_TARGET -> DOOR_DASHER_CROSS_TRANSFER_WAIT_FOR_ALIGN_DOOR_AT_TARGET_COMPLETE [bAligningDoorStarted or (config_bNoHardwareTestMode and tTimeInState>T#0.25S)] // priority 1
                DOOR_DASHER_CROSS_TRANSFER_WAIT_FOR_ALIGN_DOOR_AT_TARGET_COMPLETE -> DOOR_DASHER_CROSS_TRANSFER_WAIT_FOR_ALL_DOORDASHERS_COMPLETE [bAligningDoorComplete] // priority 1
                DOOR_DASHER_CROSS_TRANSFER_WAIT_FOR_ALL_DOORDASHERS_COMPLETE -> DOOR_DASHER_CROSS_TRANSFER_COMPLETE [rtrigSourceLeadingAndTrailingNeighborsComplete.CLK] // priority 1
                DOOR_DASHER_CROSS_TRANSFER_COMPLETE -> EndState1 [cmd_bNext] // priority 1
            END_STATE
            COMPOSITE STATE DOOR_DASHER_INLINE_TRANSFER_SEQUENCE
                START StartState5
                STATE DOOR_DASHER_INLINE_TRANSFER_START
                    entry / regStateCall(DOOR_DASHER_INLINE_TRANSFER_START, eEntry)
                    do / regStateCall(DOOR_DASHER_INLINE_TRANSFER_START, eDo)
                    exit / regStateCall(DOOR_DASHER_INLINE_TRANSFER_START, eExit)
                STATE DOOR_DASHER_INLINE_TRANSFER_DEACTIVATE_CROSS_CYLS
                    entry / regStateCall(DOOR_DASHER_INLINE_TRANSFER_DEACTIVATE_CROSS_CYLS, eEntry)
                    do / regStateCall(DOOR_DASHER_INLINE_TRANSFER_DEACTIVATE_CROSS_CYLS, eDo)
                    exit / regStateCall(DOOR_DASHER_INLINE_TRANSFER_DEACTIVATE_CROSS_CYLS, eExit)
                CHOICE ChoiceElement6_copy
                STATE DOOR_DASHER_INLINE_TRANSFER_START_SOURCE_MOTOR
                    entry / regStateCall(DOOR_DASHER_INLINE_TRANSFER_START_SOURCE_MOTOR, eEntry)
                    do / regStateCall(DOOR_DASHER_INLINE_TRANSFER_START_SOURCE_MOTOR, eDo)
                    exit / regStateCall(DOOR_DASHER_INLINE_TRANSFER_START_SOURCE_MOTOR, eExit)
                STATE DOOR_DASHER_INLINE_TRANSFER_FIND_SOURCE_EYE_RISING_EDGE
                    entry / regStateCall(DOOR_DASHER_INLINE_TRANSFER_FIND_SOURCE_EYE_RISING_EDGE, eEntry)
                    do / regStateCall(DOOR_DASHER_INLINE_TRANSFER_FIND_SOURCE_EYE_RISING_EDGE, eDo)
                    exit / regStateCall(DOOR_DASHER_INLINE_TRANSFER_FIND_SOURCE_EYE_RISING_EDGE, eExit)
                STATE DOOR_DASHER_INLINE_TRANSFER_STOP_SOURCE_MOTOR
                    entry / regStateCall(DOOR_DASHER_INLINE_TRANSFER_STOP_SOURCE_MOTOR, eEntry)
                    do / regStateCall(DOOR_DASHER_INLINE_TRANSFER_STOP_SOURCE_MOTOR, eDo)
                    exit / regStateCall(DOOR_DASHER_INLINE_TRANSFER_STOP_SOURCE_MOTOR, eExit)
                STATE DOOR_DASHER_INLINE_TRANSFER_WAIT_FOR_ALL_DOORDASHERS_READY
                    entry / regStateCall(DOOR_DASHER_INLINE_TRANSFER_WAIT_FOR_ALL_DOORDASHERS_READY, eEntry)
                    do / regStateCall(DOOR_DASHER_INLINE_TRANSFER_WAIT_FOR_ALL_DOORDASHERS_READY, eDo)
                    exit / regStateCall(DOOR_DASHER_INLINE_TRANSFER_WAIT_FOR_ALL_DOORDASHERS_READY, eExit)
                STATE DOOR_DASHER_INLINE_TRANSFER_START_MOTORS
                    entry / regStateCall(DOOR_DASHER_INLINE_TRANSFER_START_MOTORS, eEntry)
                    do / regStateCall(DOOR_DASHER_INLINE_TRANSFER_START_MOTORS, eDo)
                    exit / regStateCall(DOOR_DASHER_INLINE_TRANSFER_START_MOTORS, eExit)
                STATE DOOR_DASHER_INLINE_TRANSFER_FIND_TARGET_EYE_RISING_EDGE
                    entry / regStateCall(DOOR_DASHER_INLINE_TRANSFER_FIND_TARGET_EYE_RISING_EDGE, eEntry)
                    do / regStateCall(DOOR_DASHER_INLINE_TRANSFER_FIND_TARGET_EYE_RISING_EDGE, eDo)
                    exit / regStateCall(DOOR_DASHER_INLINE_TRANSFER_FIND_TARGET_EYE_RISING_EDGE, eExit)
                STATE DOOR_DASHER_INLINE_TRANSFER_FIND_TARGET_EYE_FALLING_EDGE
                    entry / regStateCall(DOOR_DASHER_INLINE_TRANSFER_FIND_TARGET_EYE_FALLING_EDGE, eEntry)
                    do / regStateCall(DOOR_DASHER_INLINE_TRANSFER_FIND_TARGET_EYE_FALLING_EDGE, eDo)
                    exit / regStateCall(DOOR_DASHER_INLINE_TRANSFER_FIND_TARGET_EYE_FALLING_EDGE, eExit)
                STATE DOOR_DASHER_INLINE_TRANSFER_STOP_MOTORS
                    entry / regStateCall(DOOR_DASHER_INLINE_TRANSFER_STOP_MOTORS, eEntry)
                    do / regStateCall(DOOR_DASHER_INLINE_TRANSFER_STOP_MOTORS, eDo)
                    exit / regStateCall(DOOR_DASHER_INLINE_TRANSFER_STOP_MOTORS, eExit)
                CHOICE ChoiceElement7
                STATE DOOR_DASHER_INLINE_TRANSFER_FEEDIN_DOOR_AT_TARGET
                    entry / regStateCall(DOOR_DASHER_INLINE_TRANSFER_FEEDIN_DOOR_AT_TARGET, eEntry)
                    do / regStateCall(DOOR_DASHER_INLINE_TRANSFER_FEEDIN_DOOR_AT_TARGET, eDo)
                    exit / regStateCall(DOOR_DASHER_INLINE_TRANSFER_FEEDIN_DOOR_AT_TARGET, eExit)
                STATE DOOR_DASHER_INLINE_TRANSFER_WAIT_FOR_FEEDIN_DOOR_AT_TARGET_COMPLETE
                    entry / regStateCall(DOOR_DASHER_INLINE_TRANSFER_WAIT_FOR_FEEDIN_DOOR_AT_TARGET_COMPLETE, eEntry)
                    do / regStateCall(DOOR_DASHER_INLINE_TRANSFER_WAIT_FOR_FEEDIN_DOOR_AT_TARGET_COMPLETE, eDo)
                    exit / regStateCall(DOOR_DASHER_INLINE_TRANSFER_WAIT_FOR_FEEDIN_DOOR_AT_TARGET_COMPLETE, eExit)
                STATE DOOR_DASHER_INLINE_TRANSFER_WAIT_FOR_ALL_DOORDASHERS_COMPLETE
                    entry / regStateCall(DOOR_DASHER_INLINE_TRANSFER_WAIT_FOR_ALL_DOORDASHERS_COMPLETE, eEntry)
                    do / regStateCall(DOOR_DASHER_INLINE_TRANSFER_WAIT_FOR_ALL_DOORDASHERS_COMPLETE, eDo)
                    exit / regStateCall(DOOR_DASHER_INLINE_TRANSFER_WAIT_FOR_ALL_DOORDASHERS_COMPLETE, eExit)
                STATE DOOR_DASHER_INLINE_TRANSFER_COMPLETE
                    entry / regStateCall(DOOR_DASHER_INLINE_TRANSFER_COMPLETE, eEntry)
                    do / regStateCall(DOOR_DASHER_INLINE_TRANSFER_COMPLETE, eDo)
                    exit / regStateCall(DOOR_DASHER_INLINE_TRANSFER_COMPLETE, eExit)
                END EndState3
                StartState5 -> DOOR_DASHER_INLINE_TRANSFER_START  // priority 1, on completion
                DOOR_DASHER_INLINE_TRANSFER_START -> DOOR_DASHER_INLINE_TRANSFER_DEACTIVATE_CROSS_CYLS [cmd_bNext] // priority 1
                DOOR_DASHER_INLINE_TRANSFER_DEACTIVATE_CROSS_CYLS -> ChoiceElement6_copy [bAllCrossCylsRetracted or (config_bNoHardwareTestMode and tTimeInState>T#0.25S)] // priority 1
                ChoiceElement6_copy -> DOOR_DASHER_INLINE_TRANSFER_WAIT_FOR_ALL_DOORDASHERS_READY [pdi_inlineSourceFeedEyeRisingEdge^] // priority 1
                ChoiceElement6_copy -> DOOR_DASHER_INLINE_TRANSFER_START_SOURCE_MOTOR [TRUE] // priority 2
                DOOR_DASHER_INLINE_TRANSFER_START_SOURCE_MOTOR -> DOOR_DASHER_INLINE_TRANSFER_FIND_SOURCE_EYE_RISING_EDGE [rtrigSourceMotorMoving.Q or (config_bNoHardwareTestMode and tTimeInState>T#0.25S)] // priority 1, rising edge
                DOOR_DASHER_INLINE_TRANSFER_FIND_SOURCE_EYE_RISING_EDGE -> DOOR_DASHER_INLINE_TRANSFER_STOP_SOURCE_MOTOR [rtrigInlineSourceFeedEye.Q or (config_bNoHardwareTestMode and tTimeInState>T#0.25S)] // priority 1
                DOOR_DASHER_INLINE_TRANSFER_STOP_SOURCE_MOTOR -> DOOR_DASHER_INLINE_TRANSFER_WAIT_FOR_ALL_DOORDASHERS_READY [ftrigSourceMotorMoving.Q or (config_bNoHardwareTestMode and tTimeInState>T#0.25S)] // priority 1, rising edge
                DOOR_DASHER_INLINE_TRANSFER_WAIT_FOR_ALL_DOORDASHERS_READY -> DOOR_DASHER_INLINE_TRANSFER_START_MOTORS [rtrigSourceLeadingAndTrailingNeighborsReady.Q] // priority 1, rising edge
                DOOR_DASHER_INLINE_TRANSFER_START_MOTORS -> DOOR_DASHER_INLINE_TRANSFER_FIND_TARGET_EYE_RISING_EDGE [rtrigAllTablesMotorsMoving.Q or (config_bNoHardwareTestMode and tTimeInState>T#5.25S)] // priority 1, rising edge
                DOOR_DASHER_INLINE_TRANSFER_FIND_TARGET_EYE_RISING_EDGE -> DOOR_DASHER_INLINE_TRANSFER_FIND_TARGET_EYE_FALLING_EDGE [rtrigInlineTargetFeedEyeRising.Q or (config_bNoHardwareTestMode and tTimeInState>T#0.25S)] // priority 1, rising edge
                DOOR_DASHER_INLINE_TRANSFER_FIND_TARGET_EYE_FALLING_EDGE -> DOOR_DASHER_INLINE_TRANSFER_STOP_MOTORS [ftrigInlineTargetFeedEyeFalling.Q or (config_bNoHardwareTestMode and tTimeInState>T#0.25S)] // priority 1, rising edge
                DOOR_DASHER_INLINE_TRANSFER_STOP_MOTORS -> ChoiceElement7 [ftrigAnyTablesMotorsMoving.Q or (config_bNoHardwareTestMode and tTimeInState>T#0.25S)] // priority 1, rising edge
                ChoiceElement7 -> DOOR_DASHER_INLINE_TRANSFER_WAIT_FOR_ALL_DOORDASHERS_COMPLETE [bIsTargetBufferTable] // priority 1
                ChoiceElement7 -> DOOR_DASHER_INLINE_TRANSFER_FEEDIN_DOOR_AT_TARGET [TRUE] // priority 2
                DOOR_DASHER_INLINE_TRANSFER_FEEDIN_DOOR_AT_TARGET -> DOOR_DASHER_INLINE_TRANSFER_WAIT_FOR_FEEDIN_DOOR_AT_TARGET_COMPLETE [bFeedingInDoorStarted] // priority 1
                DOOR_DASHER_INLINE_TRANSFER_WAIT_FOR_FEEDIN_DOOR_AT_TARGET_COMPLETE -> DOOR_DASHER_INLINE_TRANSFER_WAIT_FOR_ALL_DOORDASHERS_COMPLETE [bFeedingInDoorComplete] // priority 1
                DOOR_DASHER_INLINE_TRANSFER_WAIT_FOR_ALL_DOORDASHERS_COMPLETE -> DOOR_DASHER_INLINE_TRANSFER_COMPLETE [rtrigSourceLeadingAndTrailingNeighborsComplete.CLK] // priority 1
                DOOR_DASHER_INLINE_TRANSFER_COMPLETE -> EndState3 [cmd_bNext] // priority 1
            END_STATE
            STATE DOOR_DASHER_START
                entry / regStateCall(DOOR_DASHER_START, eEntry)
                do / regStateCall(DOOR_DASHER_START, eDo)
                exit / regStateCall(DOOR_DASHER_START, eExit)
            STATE DOOR_DASHER_WAIT_FOR_SOURCE_TABLE_READY
                entry / regStateCall(DOOR_DASHER_WAIT_FOR_SOURCE_TABLE_READY, eEntry)
                do / regStateCall(DOOR_DASHER_WAIT_FOR_SOURCE_TABLE_READY, eDo)
                exit / regStateCall(DOOR_DASHER_WAIT_FOR_SOURCE_TABLE_READY, eExit)
            STATE DOOR_DASHER_WAIT_FOR_SOURCE_AND_TARGET_EXTERNAL
                entry / regStateCall(DOOR_DASHER_WAIT_FOR_SOURCE_AND_TARGET_EXTERNAL, eEntry)
                do / regStateCall(DOOR_DASHER_WAIT_FOR_SOURCE_AND_TARGET_EXTERNAL, eDo)
                exit / regStateCall(DOOR_DASHER_WAIT_FOR_SOURCE_AND_TARGET_EXTERNAL, eExit)
            STATE DOOR_DASHER_CENTER_DOOR_PRE_ROTATE
                entry / regStateCall(DOOR_DASHER_CENTER_DOOR_PRE_ROTATE, eEntry)
                do / regStateCall(DOOR_DASHER_CENTER_DOOR_PRE_ROTATE, eDo)
                exit / regStateCall(DOOR_DASHER_CENTER_DOOR_PRE_ROTATE, eExit)
            CHOICE ChoiceElement5
            STATE DOOR_DASHER_ROTATE_DOOR
                entry / regStateCall(DOOR_DASHER_ROTATE_DOOR, eEntry)
                do / regStateCall(DOOR_DASHER_ROTATE_DOOR, eDo)
                exit / regStateCall(DOOR_DASHER_ROTATE_DOOR, eExit)
            STATE DOOR_DASHER_ALIGN_DOOR
                entry / regStateCall(DOOR_DASHER_ALIGN_DOOR, eEntry)
                do / regStateCall(DOOR_DASHER_ALIGN_DOOR, eDo)
                exit / regStateCall(DOOR_DASHER_ALIGN_DOOR, eExit)
            STATE DOOR_DASHER_READY_TO_TRANSFER
                entry / regStateCall(DOOR_DASHER_READY_TO_TRANSFER, eEntry)
                do / regStateCall(DOOR_DASHER_READY_TO_TRANSFER, eDo)
                exit / regStateCall(DOOR_DASHER_READY_TO_TRANSFER, eExit)
            CHOICE ChoiceElement4
            STATE DOOR_DASHER_SET_SOURCE_AND_TARGET_INTERNAL
                entry / regStateCall(DOOR_DASHER_SET_SOURCE_AND_TARGET_INTERNAL, eEntry)
                do / regStateCall(DOOR_DASHER_SET_SOURCE_AND_TARGET_INTERNAL, eDo)
                exit / regStateCall(DOOR_DASHER_SET_SOURCE_AND_TARGET_INTERNAL, eExit)
            STATE DOOR_DASHER_COMPLETE
                entry / regStateCall(DOOR_DASHER_COMPLETE, eEntry)
                do / regStateCall(DOOR_DASHER_COMPLETE, eDo)
                exit / regStateCall(DOOR_DASHER_COMPLETE, eExit)
            END EndState2
            StartState4 -> DOOR_DASHER_START  // priority 1, on completion
            DOOR_DASHER_CROSS_TRANSFER_SEQUENCE -> DOOR_DASHER_SET_SOURCE_AND_TARGET_INTERNAL  // priority 1, on completion
            DOOR_DASHER_INLINE_TRANSFER_SEQUENCE -> DOOR_DASHER_SET_SOURCE_AND_TARGET_INTERNAL  // priority 1, on completion
            DOOR_DASHER_START -> DOOR_DASHER_WAIT_FOR_SOURCE_TABLE_READY [cmd_bNext] // priority 1
            DOOR_DASHER_WAIT_FOR_SOURCE_TABLE_READY -> DOOR_DASHER_WAIT_FOR_SOURCE_AND_TARGET_EXTERNAL [bSourceTableReady] // priority 1
            DOOR_DASHER_WAIT_FOR_SOURCE_AND_TARGET_EXTERNAL -> ChoiceElement5 [bAllSourceAndTargetExternal] // priority 1
            DOOR_DASHER_CENTER_DOOR_PRE_ROTATE -> DOOR_DASHER_ROTATE_DOOR [ftrigSelfCenterComplete.Q] // priority 1, rising edge
            ChoiceElement5 -> DOOR_DASHER_CENTER_DOOR_PRE_ROTATE [cmd_bCenterDoor] // priority 1
            ChoiceElement5 -> DOOR_DASHER_ROTATE_DOOR [cmd_bRotateDoor] // priority 2
            ChoiceElement5 -> DOOR_DASHER_READY_TO_TRANSFER [TRUE] // priority 3
            DOOR_DASHER_ROTATE_DOOR -> DOOR_DASHER_ALIGN_DOOR [ftrigRotateComplete.Q] // priority 1, rising edge
            DOOR_DASHER_ALIGN_DOOR -> DOOR_DASHER_READY_TO_TRANSFER [ftrigAlignComplete.Q] // priority 1, rising edge
            DOOR_DASHER_READY_TO_TRANSFER -> ChoiceElement4 [cmd_bNext] // priority 1
            ChoiceElement4 -> DOOR_DASHER_CROSS_TRANSFER_SEQUENCE [cmd_bCrossTransfer] // priority 1
            ChoiceElement4 -> DOOR_DASHER_INLINE_TRANSFER_SEQUENCE [cmd_bInlineTransfer] // priority 2
            ChoiceElement4 -> DOOR_DASHER_SET_SOURCE_AND_TARGET_INTERNAL [TRUE] // priority 3
            DOOR_DASHER_SET_SOURCE_AND_TARGET_INTERNAL -> DOOR_DASHER_COMPLETE [not bAnyTableExternal] // priority 1
            DOOR_DASHER_COMPLETE -> EndState2 [cmd_bNext] // priority 1
        END_STATE
        StartState2 -> DOOR_DASHER_AUTOFEED_OFF  // priority 1, on completion
        DOOR_DASHER_AUTOFEED_OFF -> DOOR_DASHER_AUTOFEED_ON [cmd_bAutofeedOn] // priority 1
        DOOR_DASHER_AUTOFEED_ON -> DOOR_DASHER_DOORDASH_SEQ [cmd_bDoorDash] // priority 1, rising edge
        DOOR_DASHER_AUTOFEED_ON -> DOOR_DASHER_AUTOFEED_OFF [not cmd_bAutofeedOn] // priority 2
        DOOR_DASHER_DOORDASH_SEQ -> DOOR_DASHER_AUTOFEED_ON  // priority 1, on completion
        DOOR_DASHER_DOORDASH_SEQ -> DOOR_DASHER_AUTOFEED_OFF [ftrigAutofeedOn.Q] // priority 2, exception, rising edge
    END_STATE
    COMPOSITE STATE test
    END_STATE
    StartState1 -> DOOR_DASHER_DISABLED  // priority 1, on completion
    DOOR_DASHER_ERROR -> DOOR_DASHER_DISABLED [not cmd_bEnable] // priority 1
    DOOR_DASHER_ERROR -> DOOR_DASHER_ENABLED [cmd_bReset] / bError:=false // priority 2, rising edge
    DOOR_DASHER_DISABLED -> DOOR_DASHER_ENABLING [cmd_bEnable] // priority 1
    DOOR_DASHER_ENABLING -> DOOR_DASHER_ENABLED [downstream.status_bDownstreamAllReady] // priority 1
    DOOR_DASHER_ENABLED -> DOOR_DASHER_DISABLED [not cmd_bEnable] // priority 1, exception
    DOOR_DASHER_ENABLED -> DOOR_DASHER_ERROR [bError] // priority 2, exception
    test -> DOOR_DASHER_ENABLED [cmd_bNext] // priority 1, exception
    test -> DOOR_DASHER_ENABLED [config_bStepMode] // priority 2, exception
    test -> DOOR_DASHER_ENABLED [bAllTablesReady] // priority 3, exception
    test -> DOOR_DASHER_ENABLED [bIsConveyorAtTarget] // priority 4, exception
    test -> DOOR_DASHER_ENABLED [bIsConveyorAtSource] // priority 5, exception
    test -> DOOR_DASHER_ENABLED [bAllSourceAndTargetExternal] // priority 6, exception
    test -> DOOR_DASHER_ENABLED [status_bBusy] // priority 7, exception
    test -> DOOR_DASHER_ENABLED [bMovingFwd] // priority 8, exception
    test -> DOOR_DASHER_ENABLED [cmd_bInlineTransfer] // priority 9, exception
    test -> DOOR_DASHER_ENABLED [cmd_bCrossTransfer] // priority 10, exception
END_STATECHART
END_METHOD

METHOD feedinDoorAtTarget
IF NOT bIsConveyorAtTarget THEN
	MAIN.mainStateMachine.asmTableManagers[cmd_iTarget].smC234FeedManager.cmd_bFeedIn := TRUE;
END_IF
END_METHOD

METHOD findSourceLeadingNeighborTableIndex : INT
VAR
	iSourceLeadingNeighborTableIndex : INT;
END_VAR
findSourceLeadingNeighborTableIndex := -1;
IF bMovingFwd THEN
	IF cmd_bCrossTransfer THEN
		iSourceLeadingNeighborTableIndex := MAIN.mainStateMachine.smCtrlInterface.config_stTransferTableConfig.PrimaryTable.Tables[cmd_iSource].NeighborNorthIndex;
	ELSIF cmd_bInlineTransfer THEN
		iSourceLeadingNeighborTableIndex := MAIN.mainStateMachine.smCtrlInterface.config_stTransferTableConfig.PrimaryTable.Tables[cmd_iSource].NeighborEastIndex;
	END_IF
ELSE
	IF cmd_bCrossTransfer THEN
		iSourceLeadingNeighborTableIndex := MAIN.mainStateMachine.smCtrlInterface.config_stTransferTableConfig.PrimaryTable.Tables[cmd_iSource].NeighborSouthIndex;
	ELSIF cmd_bInlineTransfer THEN
		iSourceLeadingNeighborTableIndex := MAIN.mainStateMachine.smCtrlInterface.config_stTransferTableConfig.PrimaryTable.Tables[cmd_iSource].NeighborWestIndex;
	END_IF
END_IF
findSourceLeadingNeighborTableIndex := iSourceLeadingNeighborTableIndex;
END_METHOD

METHOD findSourceTrailingNeighborTableIndex : INT
VAR
	iSourceTrailingNeighborTableIndex : INT;
END_VAR
findSourceTrailingNeighborTableIndex := -1;
IF bMovingFwd THEN
	IF cmd_bCrossTransfer THEN
		iSourceTrailingNeighborTableIndex := MAIN.mainStateMachine.smCtrlInterface.config_stTransferTableConfig.PrimaryTable.Tables[cmd_iSource].NeighborSouthIndex;
	ELSIF cmd_bInlineTransfer THEN
		iSourceTrailingNeighborTableIndex := MAIN.mainStateMachine.smCtrlInterface.config_stTransferTableConfig.PrimaryTable.Tables[cmd_iSource].NeighborWestIndex;
	END_IF
ELSE
	IF cmd_bCrossTransfer THEN
		iSourceTrailingNeighborTableIndex := MAIN.mainStateMachine.smCtrlInterface.config_stTransferTableConfig.PrimaryTable.Tables[cmd_iSource].NeighborNorthIndex;
	ELSIF cmd_bInlineTransfer THEN
		iSourceTrailingNeighborTableIndex := MAIN.mainStateMachine.smCtrlInterface.config_stTransferTableConfig.PrimaryTable.Tables[cmd_iSource].NeighborEastIndex;
	END_IF
END_IF
findSourceTrailingNeighborTableIndex := iSourceTrailingNeighborTableIndex;
END_METHOD

METHOD findTargetPathIndex : INT
VAR_INPUT
	iSourceOrTargetIndex : INT;
END_VAR
VAR
	i : INT;
END_VAR
findTargetPathIndex := -1;
FOR i:= 0 TO pstDoorTrack^.TargetPath.PathCount - 1 DO
	IF pstDoorTrack^.TargetPath.Path[i].TableIndex = iSourceOrTargetIndex THEN
		findTargetPathIndex := i;
		RETURN;
	END_IF
END_FOR
END_METHOD

METHOD getStateDescription : STRING
CASE (machineState) OF

	DOOR_DASHER_DISABLED:
		getStateDescription := 'Disabled';
		
	DOOR_DASHER_ENABLING:
		getStateDescription := 'Enabling';
		
	DOOR_DASHER_AUTOFEED_OFF:
		getStateDescription := 'Autofeed Off';
		
	DOOR_DASHER_AUTOFEED_ON:
		getStateDescription := 'Autofeed On';
		
	DOOR_DASHER_START:
		getStateDescription := 'Starting';
			
	DOOR_DASHER_WAIT_FOR_SOURCE_TABLE_READY:
		getStateDescription := 'Wait for Source Ready';
			
	DOOR_DASHER_WAIT_FOR_SOURCE_AND_TARGET_EXTERNAL:
		getStateDescription := 'Waiting for Source and Target External';
			
	DOOR_DASHER_CENTER_DOOR_PRE_ROTATE:
		getStateDescription := 'Center Door Pre-Rotate';
			
	DOOR_DASHER_ROTATE_DOOR:
		getStateDescription := 'Rotate Door';
			
	DOOR_DASHER_ALIGN_DOOR:
		getStateDescription := 'Align Door';
			
	
	DOOR_DASHER_READY_TO_TRANSFER:
		getStateDescription := 'Ready to Transfer';
			
		
	DOOR_DASHER_CROSS_TRANSFER_START:
		getStateDescription := 'Cross Transfer Starting';
	
	DOOR_DASHER_CROSS_TRANSFER_ACTIVATE_CROSS_CYLS:
		getStateDescription := 'Activating Source and Target Cross Cylinders';


	DOOR_DASHER_CROSS_TRANSFER_START_SOURCE_MOTOR:
		getStateDescription := 'Starting Source Motor';

	DOOR_DASHER_CROSS_TRANSFER_FIND_SOURCE_EYE_RISING_EDGE:
		getStateDescription := 'Finding Source Eye Rising Edge';

	DOOR_DASHER_CROSS_TRANSFER_STOP_SOURCE_MOTOR:
		getStateDescription := 'Stopping Source Motor';
		
	DOOR_DASHER_CROSS_TRANSFER_WAIT_FOR_ALL_DOORDASHERS_READY:
		getStateDescription := 'Waiting for All Door Dashers Ready';
		
	DOOR_DASHER_CROSS_TRANSFER_START_MOTORS:
		getStateDescription := 'Starting Motors';
	
	DOOR_DASHER_CROSS_TRANSFER_FIND_TARGET_EYE_RISING_EDGE_PRE:
		getStateDescription := 'Finding Target Eye Rising Edge - Pre';
			
	DOOR_DASHER_CROSS_TRANSFER_FIND_TARGET_EYE_RISING_EDGE_POST:
		getStateDescription := 'Finding (Conveyor) Target Eye Rising Edge - POST';
	
	DOOR_DASHER_CROSS_TRANSFER_FIND_RISING_OR_FALLING_EDGE_OF_TARGET_EYE:
		getStateDescription := 'Finding (Non-Conveyor) Target Eye';
	
	DOOR_DASHER_CROSS_TRANSFER_STOP_MOTORS:
		getStateDescription := 'Stopping Motors';
		
	DOOR_DASHER_CROSS_TRANSFER_RESTART_TARGET_MOTOR:
		getStateDescription := 'Restarting Target and Reverse Direction for Wide Door';
	
	DOOR_DASHER_CROSS_TRANSFER_FIND_RISING_EDGE_OF_TARGET_FENCE_EYE:
		getStateDescription := 'Finding Rising Edge of Target-Fence Eye';
		
	DOOR_DASHER_CROSS_TRANSFER_STOP_MOTORS_ON_TARGET_FENCE_EYE:
		getStateDescription := 'Stopping Motors on Target Fence Eye';
		
	DOOR_DASHER_CROSS_TRANSFER_DEACTIVATE_CROSS_CYLS:
		getStateDescription := 'Deactivating Cross Cylinders';
		
	DOOR_DASHER_CROSS_TRANSFER_ALIGN_DOOR_AT_TARGET:
		getStateDescription := 'Aligning Door at Target';
		
	DOOR_DASHER_CROSS_TRANSFER_WAIT_FOR_ALIGN_DOOR_AT_TARGET_COMPLETE:
		getStateDescription := 'Wait for Align Door at Target Complete';
		
	DOOR_DASHER_CROSS_TRANSFER_WAIT_FOR_ALL_DOORDASHERS_COMPLETE:
		getStateDescription := 'Wait for All Door Dashers Complete';
	
	DOOR_DASHER_CROSS_TRANSFER_COMPLETE:
		getStateDescription := 'Cross Transfer Complete';
		
	DOOR_DASHER_SET_SOURCE_AND_TARGET_INTERNAL:
		getStateDescription := 'Setting Source and Target in Internal State';
	
	DOOR_DASHER_COMPLETE:
		getStateDescription := 'Door Dasher Complete';
	
	DOOR_DASHER_INLINE_TRANSFER_START:
		getStateDescription := 'Inline Transfer Starting';
	
	DOOR_DASHER_INLINE_TRANSFER_DEACTIVATE_CROSS_CYLS:
		getStateDescription := 'Deactivating Source and Target Cross Cylinders';
		
	DOOR_DASHER_INLINE_TRANSFER_START_SOURCE_MOTOR:
		getStateDescription := 'Starting Source Motor';
		
	DOOR_DASHER_INLINE_TRANSFER_FIND_SOURCE_EYE_RISING_EDGE:
		getStateDescription := 'Finding Source Eye Rising Edge';
		
	DOOR_DASHER_INLINE_TRANSFER_STOP_SOURCE_MOTOR:
		getStateDescription := 'Stopping Source Motor';
		
	DOOR_DASHER_INLINE_TRANSFER_WAIT_FOR_ALL_DOORDASHERS_READY:
		getStateDescription := 'Waiting for All Door Dashers Ready';
		
	DOOR_DASHER_INLINE_TRANSFER_START_MOTORS:
		getStateDescription := 'Starting Motors';
		
	DOOR_DASHER_INLINE_TRANSFER_FIND_TARGET_EYE_RISING_EDGE:
		getStateDescription := 'Finding Target Eye Rising Edge';
		
	DOOR_DASHER_INLINE_TRANSFER_FIND_TARGET_EYE_FALLING_EDGE:
		getStateDescription := 'Finding Target Eye Falling Edge';
		
	DOOR_DASHER_INLINE_TRANSFER_STOP_MOTORS:
		getStateDescription := 'Stopping Motors';
		
	DOOR_DASHER_INLINE_TRANSFER_FEEDIN_DOOR_AT_TARGET:
		getStateDescription := 'Feedin Door at Target';
		
	DOOR_DASHER_INLINE_TRANSFER_WAIT_FOR_FEEDIN_DOOR_AT_TARGET_COMPLETE:
		getStateDescription := 'Wait for Feedin Door at Target Complete';
		
	DOOR_DASHER_INLINE_TRANSFER_WAIT_FOR_ALL_DOORDASHERS_COMPLETE:
		getStateDescription := 'Wait for All Door Dashers Complete';
		
	DOOR_DASHER_INLINE_TRANSFER_COMPLETE:
		getStateDescription := 'Inline Transfer Complete';
		
	DOOR_DASHER_ERROR:
		getStateDescription := 'Error';
		
END_CASE

IF status_bBusy THEN
	fbTaskMaster.fbFormatString(sFormat:='[%s->%s] ', 
		arg1:= F_STRINGEX(sSource),
		arg2:= F_STRINGEX(sTarget));
	getStateDescription := concat(fbTaskMaster.fbFormatString.sOut, getStateDescription);
END_IF

// Call this last to pick up any unassigned descriptions
SUPER^.getStateDescription();
END_METHOD

METHOD getTableName : STRING
VAR_INPUT
	tableIndex : INT;
END_VAR
IF tableIndex >= 0 AND tableIndex < MAX_TABLES_COUNT THEN
	getTableName := MAIN.mainStateMachine.smCtrlInterface.config_stTransferTableConfig.PrimaryTable.Tables[tableIndex].Name;
ELSE
	getTableName := '---';
END_IF
END_METHOD

METHOD goFast
VAR 
	i : INT;
	tableIndex : INT;
END_VAR
FOR i:=iSourcePathIndex TO iTargetPathIndex DO
	tableIndex := stTargetPath.Path[i].TableIndex;
	MAIN.mainStateMachine.asmTableManagers[tableIndex].psmHcFeedMotor^.cmd_iSpeedRPM := MAIN.mainStateMachine.asmTableManagers[tableIndex].iFeedFastSpeedRPM;
END_FOR
END_METHOD

METHOD goFwd
VAR 
	i : INT;
	tableIndex : INT;
END_VAR
FOR i:=iSourcePathIndex TO iTargetPathIndex DO
	tableIndex := stTargetPath.Path[i].TableIndex;
	MAIN.mainStateMachine.asmTableManagers[tableIndex].goFwd();
END_FOR
END_METHOD

METHOD goRev
VAR 
	i : INT;
	tableIndex : INT;
END_VAR
FOR i:=iSourcePathIndex TO iTargetPathIndex DO
	tableIndex := stTargetPath.Path[i].TableIndex;
	MAIN.mainStateMachine.asmTableManagers[tableIndex].goRev();
END_FOR
END_METHOD

METHOD goSlow
VAR 
	i : INT;
	tableIndex : INT;
END_VAR
FOR i:=iSourcePathIndex TO iTargetPathIndex DO
	tableIndex := stTargetPath.Path[i].TableIndex;
	MAIN.mainStateMachine.asmTableManagers[tableIndex].psmHcFeedMotor^.cmd_iSpeedRPM := MAIN.mainStateMachine.asmTableManagers[tableIndex].iFeedSlowSpeedRPM;
END_FOR
END_METHOD

METHOD initialize
SUPER^.initialize();		// must run first
descriptor.sModuleClass := 'Door Dasher';
END_METHOD

METHOD inlineTransferStart
tFindTargetEyeTimeout := LREAL_TO_TIME((ABS(iSourcePathIndex - iTargetPathIndex) * config_fFindTargetEyeTimeSec) * 1000);
sSource := getTableName(cmd_iSource);
sTarget := getTableName(cmd_iTarget);
bDoorInMachineAtSource		:= MAIN.mainStateMachine.asmTableManagers[cmd_iSource].bDoorInMachine;
bDoorInMachineAtTarget		:= MAIN.mainStateMachine.asmTableManagers[cmd_iTarget].bDoorInMachine;
MAIN.mainStateMachine.asmTableManagers[cmd_iSource].setTransferOutStarted();
MAIN.mainStateMachine.asmTableManagers[cmd_iTarget].setDoorTransferredInStarted();
bIsTargetBufferTable := MAIN.mainStateMachine.asmTableManagers[cmd_iTarget].config_bIsBufferTable;

IF bMovingFwd THEN
	pdi_inlineSourceFeedEyeRisingEdge := ADR( MAIN.mainStateMachine.asmTableManagers[cmd_iSource].smC234FeedManager.di_BSideDoorSenseEye);
	pdi_inlineTargetFeedEyeRisingEdge := ADR( MAIN.mainStateMachine.asmTableManagers[cmd_iTarget].smC234FeedManager.di_ASideDoorSenseEye);
	pdi_inlineTargetFeedEyeFallingEdge := ADR( MAIN.mainStateMachine.asmTableManagers[cmd_iTarget].smC234FeedManager.di_ASideDoorSenseEye);
ELSE
	pdi_inlineSourceFeedEyeRisingEdge := ADR( MAIN.mainStateMachine.asmTableManagers[cmd_iSource].smC234FeedManager.di_ASideDoorSenseEye);
	pdi_inlineTargetFeedEyeRisingEdge := ADR( MAIN.mainStateMachine.asmTableManagers[cmd_iTarget].smC234FeedManager.di_BSideDoorSenseEye);
	pdi_inlineTargetFeedEyeFallingEdge := ADR( MAIN.mainStateMachine.asmTableManagers[cmd_iTarget].smC234FeedManager.di_BSideDoorSenseEye);
END_IF
END_METHOD

METHOD isAligningDoorAtTarget : BOOL
isAligningDoorAtTarget := TRUE;
IF NOT bIsConveyorAtTarget THEN
	isAligningDoorAtTarget := MAIN.mainStateMachine.asmTableManagers[cmd_iTarget].smC234FeedManager.bAlignRunning;
END_IF
END_METHOD

METHOD isAligningDoorAtTargetComplete : BOOL
isAligningDoorAtTargetComplete := TRUE;
IF NOT bIsConveyorAtTarget THEN
	isAligningDoorAtTargetComplete := NOT MAIN.mainStateMachine.asmTableManagers[cmd_iTarget].smC234FeedManager.bAlignRunning;
END_IF
END_METHOD

METHOD isFeedingInDoorAtTarget : BOOL
IF NOT bIsConveyorAtTarget THEN
	isFeedingInDoorAtTarget := MAIN.mainStateMachine.asmTableManagers[cmd_iTarget].smC234FeedManager.bFeedinRunning;
END_IF
END_METHOD

METHOD isFeedingInDoorAtTargetComplete : BOOL
IF NOT bIsConveyorAtTarget THEN
	isFeedingInDoorAtTargetComplete := 
		NOT (MAIN.mainStateMachine.asmTableManagers[cmd_iTarget].smC234FeedManager.bFeedinRunning OR
		 MAIN.mainStateMachine.asmTableManagers[cmd_iTarget].smC234FeedManager.bAlignRunning OR
		 MAIN.mainStateMachine.asmTableManagers[cmd_iTarget].smC234FeedManager.status_bBusy);
END_IF
END_METHOD

METHOD isSourceLeadingNeighborComplete : BOOL
VAR_INPUT
END_VAR
IF iSourceLeadingNeighborIndex = -1 THEN
	isSourceLeadingNeighborComplete := TRUE;
	RETURN;
END_IF

IF NOT MAIN.mainStateMachine.asmTableManagers[iSourceLeadingNeighborIndex].bHasDoor THEN
	isSourceLeadingNeighborComplete := TRUE;
	RETURN;
END_IF

// At this point, the 'leading' neighbor has a door.
IF NOT (MAIN.mainStateMachine.asmTableManagers[iSourceLeadingNeighborIndex].smDoorDasher.bCrossTransferSeqRunning OR 
	MAIN.mainStateMachine.asmTableManagers[iSourceLeadingNeighborIndex].smDoorDasher.bInlineTransferSeqRunning) THEN
	isSourceLeadingNeighborComplete := TRUE;
	RETURN;
END_IF

// At this point, the 'leading' neighbor has a door and its DoorDasher's transferring seq is running.


// Finally, the source leading neighbor is complete if both the source's and the leading neighbor has door are going in the same direction.
isSourceLeadingNeighborComplete := 
	(MAIN.mainStateMachine.asmTableManagers[iSourceLeadingNeighborIndex].smDoorDasher.bCrossTransferWaitingForAllDoorDashersComplete OR 
	 MAIN.mainStateMachine.asmTableManagers[iSourceLeadingNeighborIndex].smDoorDasher.bInlineTransferWaitingForAllDoorDashersComplete) AND
	stCurrentTargetNode.Direction = eSourceLeadingNeighborNodeDirection;
END_METHOD

METHOD isSourceLeadingNeighborReady : BOOL
VAR_INPUT
END_VAR
IF iSourceLeadingNeighborIndex = -1 THEN
	isSourceLeadingNeighborReady := TRUE;
	RETURN;
END_IF

IF NOT MAIN.mainStateMachine.asmTableManagers[iSourceLeadingNeighborIndex].bHasDoor THEN
	isSourceLeadingNeighborReady := TRUE;
	RETURN;
END_IF

// At this point, the 'leading' neighbor has a door.
IF NOT (MAIN.mainStateMachine.asmTableManagers[iSourceLeadingNeighborIndex].smDoorDasher.bCrossTransferSeqRunning OR 
	MAIN.mainStateMachine.asmTableManagers[iSourceLeadingNeighborIndex].smDoorDasher.bInlineTransferSeqRunning) THEN
	isSourceLeadingNeighborReady := TRUE;
	RETURN;
END_IF

// At this point, the 'leading' neighbor has a door and its DoorDasher's transferring seq is running.


// Finally, the source leading neighbor is ready if both the source's and the leading neighbor has door are going in the same direction.
isSourceLeadingNeighborReady := 
	(MAIN.mainStateMachine.asmTableManagers[iSourceLeadingNeighborIndex].smDoorDasher.bCrossTransferWaitingForAllDoorDashersReady OR 
	 MAIN.mainStateMachine.asmTableManagers[iSourceLeadingNeighborIndex].smDoorDasher.bInlineTransferWaitingForAllDoorDashersReady) AND
	stCurrentTargetNode.Direction = eSourceLeadingNeighborNodeDirection;
END_METHOD

METHOD isSourceMotorMoving : BOOL
VAR 
	tableIndex : INT;
END_VAR
tableIndex := stTargetPath.Path[iSourcePathIndex].TableIndex;
isSourceMotorMoving := MAIN.mainStateMachine.asmTableManagers[tableIndex].status_bMoving;
END_METHOD

METHOD isSourceTableReady : BOOL
VAR 
	tableIndex : INT;
END_VAR
tableIndex := stTargetPath.Path[iSourcePathIndex].TableIndex;
isSourceTableReady := 
	NOT (MAIN.mainStateMachine.asmTableManagers[tableIndex].anyChildBusy()
	) AND 
	MAIN.mainStateMachine.asmTableManagers[tableIndex].cmd_bAutoFeedOn;
END_METHOD

METHOD isSourceTrailingNeighborComplete : BOOL
VAR_INPUT
END_VAR
IF iSourceTrailingNeighborIndex = -1 THEN
	isSourceTrailingNeighborComplete := TRUE;
	RETURN;
END_IF

IF NOT MAIN.mainStateMachine.asmTableManagers[iSourceTrailingNeighborIndex].bHasDoor THEN
	isSourceTrailingNeighborComplete := TRUE;
	RETURN;
END_IF

// At this point, the 'trailing' neighbor has a door.
IF NOT (MAIN.mainStateMachine.asmTableManagers[iSourceTrailingNeighborIndex].smDoorDasher.bCrossTransferSeqRunning OR 
	MAIN.mainStateMachine.asmTableManagers[iSourceTrailingNeighborIndex].smDoorDasher.bInlineTransferSeqRunning) THEN
	isSourceTrailingNeighborComplete := TRUE;
	RETURN;
END_IF

// At this point, the 'trailing' neighbor has a door and its DoorDasher's transferring seq is running.

// Finally, check if the source's trailing neighbor is complete.
isSourceTrailingNeighborComplete := 
	stCurrentTargetNode.Direction <> MAIN.mainStateMachine.asmTableManagers[iSourceTrailingNeighborIndex].smDoorDasher.stCurrentTargetNode.Direction OR // TODO: if the source's trailing neighbor is not moving in the same direction, then it's considered complete.
	(MAIN.mainStateMachine.asmTableManagers[iSourceTrailingNeighborIndex].smDoorDasher.bCrossTransferWaitingForAllDoorDashersComplete OR 
	 MAIN.mainStateMachine.asmTableManagers[iSourceTrailingNeighborIndex].smDoorDasher.bInlineTransferWaitingForAllDoorDashersComplete)
	;
END_METHOD

METHOD isSourceTrailingNeighborReady : BOOL
VAR_INPUT
END_VAR
IF iSourceTrailingNeighborIndex = -1 THEN
	isSourceTrailingNeighborReady := TRUE;
	RETURN;
END_IF

IF NOT MAIN.mainStateMachine.asmTableManagers[iSourceTrailingNeighborIndex].bHasDoor THEN
	isSourceTrailingNeighborReady := TRUE;
	RETURN;
END_IF

// At this point, the 'trailing' neighbor has a door.
IF NOT (MAIN.mainStateMachine.asmTableManagers[iSourceTrailingNeighborIndex].smDoorDasher.bCrossTransferSeqRunning OR 
	MAIN.mainStateMachine.asmTableManagers[iSourceTrailingNeighborIndex].smDoorDasher.bInlineTransferSeqRunning) THEN
	isSourceTrailingNeighborReady := TRUE;
	RETURN;
END_IF

// At this point, the 'trailing' neighbor has a door and its DoorDasher's transferring seq is running.

// Finally, check if the source's trailing neighbor is ready.
isSourceTrailingNeighborReady := 
	stCurrentTargetNode.Direction <> MAIN.mainStateMachine.asmTableManagers[iSourceTrailingNeighborIndex].smDoorDasher.stCurrentTargetNode.Direction OR // TODO: if the source's trailing neighbor is not moving in the same direction, then it's considered ready.
	(MAIN.mainStateMachine.asmTableManagers[iSourceTrailingNeighborIndex].smDoorDasher.bCrossTransferWaitingForAllDoorDashersReady OR 
	 MAIN.mainStateMachine.asmTableManagers[iSourceTrailingNeighborIndex].smDoorDasher.bInlineTransferWaitingForAllDoorDashersReady)
	;
END_METHOD

METHOD isTargetMotorMoving : BOOL
VAR 
	tableIndex : INT;
END_VAR
tableIndex := stTargetPath.Path[iTargetPathIndex].TableIndex;
isTargetMotorMoving := MAIN.mainStateMachine.asmTableManagers[tableIndex].status_bMoving;
END_METHOD

METHOD isTargetTransferTableCandDsideDoorFeedEyesClear : BOOL
VAR_INPUT
END_VAR
isTargetTransferTableCandDsideDoorFeedEyesClear := 
	bIsConveyorAtTarget OR
	NOT (MAIN.mainStateMachine.asmTableManagers[cmd_iTarget].smC234FeedManager.di_CSideDoorFeedEye OR
		MAIN.mainStateMachine.asmTableManagers[cmd_iTarget].smC234FeedManager.di_DSideDoorFeedEye);
END_METHOD

METHOD postProcess
VAR_INPUT
END_VAR
SUPER^.postProcess();
cmd_bReset := FALSE;
cmd_bDoorDash := FALSE;
END_METHOD

(* this method is run before the doState is run*)
METHOD preProcess
SUPER^.preProcess();

bCrossTransferWaitingForAllDoorDashersReady := machineState = DOOR_DASHER_CROSS_TRANSFER_WAIT_FOR_ALL_DOORDASHERS_READY;
bCrossTransferWaitingForAllDoorDashersComplete := machineState = DOOR_DASHER_CROSS_TRANSFER_WAIT_FOR_ALL_DOORDASHERS_COMPLETE;

bInlineTransferWaitingForAllDoorDashersReady := machineState = DOOR_DASHER_INLINE_TRANSFER_WAIT_FOR_ALL_DOORDASHERS_READY;
bInlineTransferWaitingForAllDoorDashersComplete := machineState = DOOR_DASHER_INLINE_TRANSFER_WAIT_FOR_ALL_DOORDASHERS_COMPLETE;

ftrigAutofeedOn(CLK:=cmd_bAutoFeedOn);

IF iErrorId <> 0 THEN
	raiseError(FALSE);
END_IF


IF NOT cmd_bEnable THEN
	IF machineState > DOOR_DASHER_ENABLING AND
		machineState <= DOOR_DASHER_ERROR THEN
		machineState := DOOR_DASHER_DISABLED;
	END_IF	
ELSIF bError THEN
	IF machineState > DOOR_DASHER_ENABLING AND
		machineState < DOOR_DASHER_ERROR THEN
		machineState := DOOR_DASHER_ERROR;
	END_IF
ELSIF ftrigAutofeedOn.Q THEN
	IF machineState > DOOR_DASHER_AUTOFEED_OFF AND
		machineState < DOOR_DASHER_ERROR THEN
		machineState := DOOR_DASHER_AUTOFEED_OFF;
	END_IF
END_IF
END_METHOD

